KUKA KRL program: EPS_2_251455_MH64A_A_20251003045107.src

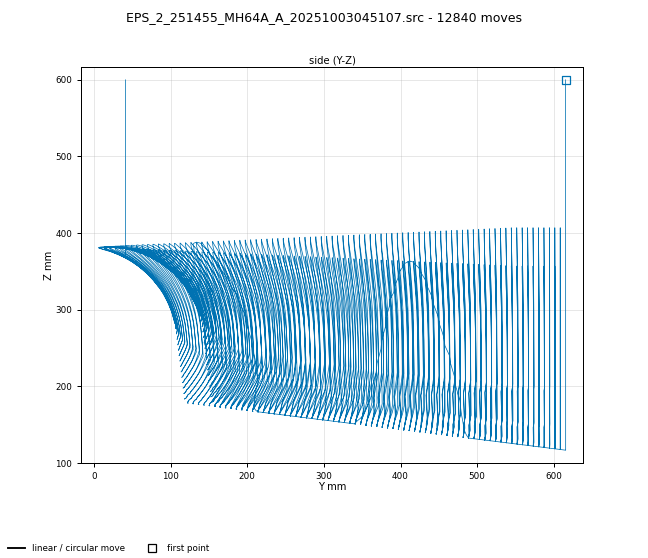
[picture p0: tool path of EPS_2_251455_MH64A_A_20251003045107.src, 12840 of 12842 moves have a stored position in this frame; points joined in program order, loops and branches not executed]
&ACCESS RVP
&REL 4
&COMMENT QRS 19112012
&PARAM EDITMASK = *
DEF PART()
EXT BAS (BAS_COMMAND :IN,REAL :IN )
INT I
BAS (#INITMOV,0 )

;KUKA QRS Post kuka4.cps  Date:22-06-2017 !

File_ID=2880

QRS_PRE_INIT()

;Init var - Until changes are made in qrs_pre_init
Outlet_Square_prg=0
Inlet_1_Square_prg=0
Inlet_2_Square_prg=0
Inlet_3_Square_prg=0
Inlet_4_Square_prg=0
Inlet_5_Square_prg=0

Outlet_1={X 0.000, Y 546.330, Z 306.500, B 0.000, E1 0.000 }
Inlet_1={X 0.000, Y 549.890, Z 256.500, B 0.000, E1 175.000 }
Outlet_1_type=201
Inlet_1_type=201
;QRS#1=Sidecore dimensions
;QRS#2=200-8" PVC SDR 35
;QRS#3=200-8" PVC SDR 35
;QRS#4=
;QRS#5=
;QRS#6=
;QRS#7=
;QRS#8=
;QRS#9=12-08 PSX
;QRS#10=12-08 PSX
;QRS#11=
;QRS#12=
;QRS#13=
;QRS#14=
;QRS#15=
;QRS#16=1220x127x686 2,25'
;QRS#17=EPS Height
;QRS#18=407
;QRS#19=*
;QRS#20= UPDATED VERSION 22-06-2017
;QRS#21=*
Outlet_Square=0100
Inlet_1_Square=0100
Inlet_2_Square=0
Inlet_3_Square=0
Inlet_4_Square=0
Inlet_5_Square=0
Mill_Square=1
Outlet_Square_Prg=204
Inlet_1_Square_prg=204

QRS_INIT()

$ADVANCE=5

; T1
PTP {E1 173.652,E2 173.652}
PTP {X 0,Y 615.443,A -85,B 0,C 180,E1 173.652,E2 173.652,E3 0,E4 0,E5 0,E6 0}
QRS_SPEED_INIT()
LIN {X 0,Y 615.443,Z 600,A -85,B 0,C 180,E1 173.652,E2 173.652,E3 0,E4 0,E5 0,E6 0} C_VEL
LIN {X 0,Y 615.443,Z 126.875,A -85,B 0,C 180,E1 173.652,E2 173.652} C_VEL
LIN {X 0,Y 615.443,Z 118.696,A -85,B 0,C 180,E1 173.652,E2 173.652} C_VEL
LIN {X 0,Y 615.432,Z 116.696,A -85,B 0,C 180,E1 173.465,E2 173.465} C_VEL
LIN {X 0,Y 615.432,Z 116.696,A -85,B 0,C 180,E1 171.462,E2 171.462} C_VEL
LIN {X 0,Y 615.436,Z 116.697,A -85,B 0,C 180,E1 169.136,E2 169.136} C_VEL
LIN {X 0,Y 615.468,Z 116.699,A -85,B 0,C 180,E1 166.798,E2 166.798} C_VEL
LIN {X 0,Y 615.467,Z 116.692,A -85,B 0,C 180,E1 164.094,E2 164.094} C_VEL
LIN {X 0,Y 615.458,Z 116.692,A -85,B 0,C 180,E1 162.042,E2 162.042} C_VEL
LIN {X 0,Y 615.45,Z 116.692,A -85,B 0,C 180,E1 159.966,E2 159.966} C_VEL
LIN {X 0,Y 615.442,Z 116.694,A -85,B 0,C 180,E1 157.664,E2 157.664} C_VEL
LIN {X 0,Y 615.491,Z 116.7,A -85,B 0,C 180,E1 155.008,E2 155.008} C_VEL
LIN {X 0,Y 615.495,Z 116.694,A -85,B 0,C 180,E1 152.823,E2 152.823} C_VEL
LIN {X 0,Y 615.456,Z 116.69,A -85,B 0,C 180,E1 150.21,E2 150.21} C_VEL
LIN {X 0,Y 615.457,Z 116.696,A -85,B 0,C 180,E1 147.674,E2 147.674} C_VEL
LIN {X 0,Y 615.496,Z 116.697,A -85,B 0,C 180,E1 145.185,E2 145.185} C_VEL
LIN {X 0,Y 615.489,Z 116.686,A -85,B 0,C 180,E1 142.758,E2 142.758} C_VEL
LIN {X 0,Y 615.454,Z 116.692,A -85,B 0,C 180,E1 140.247,E2 140.247} C_VEL
LIN {X 0,Y 615.489,Z 116.699,A -85,B 0,C 180,E1 137.647,E2 137.647} C_VEL
LIN {X 0,Y 615.492,Z 116.684,A -85,B 0,C 180,E1 134.932,E2 134.932} C_VEL
LIN {X 0,Y 615.47,Z 116.696,A -85,B 0,C 180,E1 132.078,E2 132.078} C_VEL
LIN {X 0,Y 615.493,Z 116.683,A -85,B 0,C 180,E1 129.062,E2 129.062} C_VEL
LIN {X 0,Y 615.467,Z 116.693,A -85,B 0,C 180,E1 126.426,E2 126.426} C_VEL
LIN {X 0,Y 615.485,Z 116.688,A -85,B 0,C 180,E1 123.533,E2 123.533} C_VEL
LIN {X 0,Y 615.473,Z 116.687,A -85,B 0,C 180,E1 120.921,E2 120.921} C_VEL
LIN {X 0,Y 615.481,Z 116.696,A -85,B 0,C 180,E1 118.448,E2 118.448} C_VEL
LIN {X 0,Y 615.487,Z 116.684,A -85,B 0,C 180,E1 115.568,E2 115.568} C_VEL
LIN {X 0,Y 615.474,Z 116.751,A -85,B 0,C 180,E1 112.979,E2 112.979} C_VEL
LIN {X 0,Y 615.47,Z 132.079,A -85,B 0,C 180,E1 110.294,E2 110.294} C_VEL
LIN {X 0,Y 615.477,Z 146.431,A -85,B 0,C 180,E1 107.807,E2 107.807} C_VEL
LIN {X 0,Y 615.434,Z 252.88,A -85,B 0,C 180,E1 106.545,E2 106.545} C_VEL
LIN {X 0,Y 615.441,Z 266.052,A -85,B 0,C 180,E1 106.255,E2 106.255} C_VEL
LIN {X 0,Y 615.481,Z 279.193,A -85,B 0,C 180,E1 105.821,E2 105.821} C_VEL
LIN {X 0,Y 615.47,Z 290.561,A -85,B 0,C 180,E1 105.312,E2 105.312} C_VEL
LIN {X 0,Y 615.475,Z 302.26,A -85,B 0,C 180,E1 104.634,E2 104.634} C_VEL
LIN {X 0,Y 615.498,Z 312.734,A -85,B 0,C 180,E1 103.874,E2 103.874} C_VEL
LIN {X 0,Y 615.497,Z 322.104,A -85,B 0,C 180,E1 103.034,E2 103.034} C_VEL
LIN {X 0,Y 615.497,Z 331.132,A -85,B 0,C 180,E1 102.028,E2 102.028} C_VEL
LIN {X 0,Y 615.497,Z 337.241,A -85,B 0,C 180,E1 101.193,E2 101.193} C_VEL
LIN {X 0,Y 615.497,Z 343.213,A -85,B 0,C 180,E1 100.195,E2 100.195} C_VEL
LIN {X 0,Y 615.496,Z 347.904,A -85,B 0,C 180,E1 99.199,E2 99.199} C_VEL
LIN {X 0,Y 615.496,Z 351.467,A -85,B 0,C 180,E1 98.206,E2 98.206} C_VEL
LIN {X 0,Y 615.496,Z 354.018,A -85,B 0,C 180,E1 97.216,E2 97.216} C_VEL
LIN {X 0,Y 615.495,Z 355.21,A -85,B 0,C 180,E1 96.557,E2 96.557} C_VEL
LIN {X 0,Y 615.499,Z 355.969,A -85,B 0,C 180,E1 95.899,E2 95.899} C_VEL
LIN {X 0,Y 615.498,Z 356.306,A -85,B 0,C 180,E1 94.585,E2 94.585} C_VEL
LIN {X 0,Y 615.497,Z 355.907,A -85,B 0,C 180,E1 93.929,E2 93.929} C_VEL
LIN {X 0,Y 615.496,Z 353.854,A -85,B 0,C 180,E1 92.618,E2 92.618} C_VEL
LIN {X 0,Y 615.498,Z 351.251,A -85,B 0,C 180,E1 91.636,E2 91.636} C_VEL
LIN {X 0,Y 615.496,Z 347.662,A -85,B 0,C 180,E1 90.655,E2 90.655} C_VEL
LIN {X 0,Y 615.495,Z 342.984,A -85,B 0,C 180,E1 89.673,E2 89.673} C_VEL
LIN {X 0,Y 615.497,Z 335.969,A -85,B 0,C 180,E1 88.528,E2 88.528} C_VEL
LIN {X 0,Y 615.496,Z 328.361,A -85,B 0,C 180,E1 87.547,E2 87.547} C_VEL
LIN {X 0,Y 615.498,Z 318.831,A -85,B 0,C 180,E1 86.564,E2 86.564} C_VEL
LIN {X 0,Y 615.498,Z 309.005,A -85,B 0,C 180,E1 85.744,E2 85.744} C_VEL
LIN {X 0,Y 615.461,Z 297.922,A -85,B 0,C 180,E1 85.006,E2 85.006} C_VEL
LIN {X 0,Y 615.479,Z 287.084,A -85,B 0,C 180,E1 84.431,E2 84.431} C_VEL
LIN {X 0,Y 615.476,Z 275.241,A -85,B 0,C 180,E1 83.942,E2 83.942} C_VEL
LIN {X 0,Y 615.447,Z 263.329,A -85,B 0,C 180,E1 83.582,E2 83.582} C_VEL
LIN {X 0,Y 615.441,Z 249.767,A -85,B 0,C 180,E1 83.32,E2 83.32} C_VEL
LIN {X 0,Y 615.485,Z 146.439,A -85,B 0,C 180,E1 82.104,E2 82.104} C_VEL
LIN {X 0,Y 615.49,Z 130.22,A -85,B 0,C 180,E1 79.294,E2 79.294} C_VEL
LIN {X 0,Y 615.467,Z 116.69,A -85,B 0,C 180,E1 76.883,E2 76.883} C_VEL
LIN {X 0,Y 615.489,Z 116.688,A -85,B 0,C 180,E1 74.096,E2 74.096} C_VEL
LIN {X 0,Y 615.468,Z 116.696,A -85,B 0,C 180,E1 71.354,E2 71.354} C_VEL
LIN {X 0,Y 615.49,Z 116.683,A -85,B 0,C 180,E1 68.569,E2 68.569} C_VEL
LIN {X 0,Y 615.484,Z 116.699,A -85,B 0,C 180,E1 65.729,E2 65.729} C_VEL
LIN {X 0,Y 615.466,Z 116.688,A -85,B 0,C 180,E1 62.96,E2 62.96} C_VEL
LIN {X 0,Y 615.494,Z 116.696,A -85,B 0,C 180,E1 60.205,E2 60.205} C_VEL
LIN {X 0,Y 615.457,Z 116.693,A -85,B 0,C 180,E1 57.542,E2 57.542} C_VEL
LIN {X 0,Y 615.463,Z 116.689,A -85,B 0,C 180,E1 55.185,E2 55.185} C_VEL
LIN {X 0,Y 615.496,Z 116.687,A -85,B 0,C 180,E1 52.76,E2 52.76} C_VEL
LIN {X 0,Y 615.457,Z 116.695,A -85,B 0,C 180,E1 49.915,E2 49.915} C_VEL
LIN {X 0,Y 615.449,Z 116.692,A -85,B 0,C 180,E1 47.645,E2 47.645} C_VEL
LIN {X 0,Y 615.497,Z 116.688,A -85,B 0,C 180,E1 44.934,E2 44.934} C_VEL
LIN {X 0,Y 615.449,Z 116.695,A -85,B 0,C 180,E1 42.078,E2 42.078} C_VEL
LIN {X 0,Y 615.444,Z 116.693,A -85,B 0,C 180,E1 39.754,E2 39.754} C_VEL
LIN {X 0,Y 615.49,Z 116.698,A -85,B 0,C 180,E1 36.939,E2 36.939} C_VEL
LIN {X 0,Y 615.439,Z 116.694,A -85,B 0,C 180,E1 34.025,E2 34.025} C_VEL
LIN {X 0,Y 615.487,Z 116.7,A -85,B 0,C 180,E1 31.088,E2 31.088} C_VEL
LIN {X 0,Y 615.439,Z 116.697,A -85,B 0,C 180,E1 28.445,E2 28.445} C_VEL
LIN {X 0,Y 615.435,Z 116.697,A -85,B 0,C 180,E1 26.447,E2 26.447} C_VEL
LIN {X 0,Y 615.442,Z 116.694,A -85,B 0,C 180,E1 24.002,E2 24.002} C_VEL
LIN {X 0,Y 615.498,Z 116.696,A -85,B 0,C 180,E1 21.432,E2 21.432} C_VEL
LIN {X 0,Y 615.427,Z 116.697,A -85,B 0,C 180,E1 18.592,E2 18.592} C_VEL
LIN {X 0,Y 615.464,Z 116.695,A -85,B 0,C 180,E1 15.906,E2 15.906} C_VEL
LIN {X 0,Y 615.449,Z 116.699,A -85,B 0,C 180,E1 13.202,E2 13.202} C_VEL
LIN {X 0,Y 615.422,Z 116.699,A -85,B 0,C 180,E1 10.864,E2 10.864} C_VEL
LIN {X 0,Y 615.423,Z 116.699,A -85,B 0,C 180,E1 8.538,E2 8.538} C_VEL
LIN {X 0,Y 615.496,Z 116.698,A -85,B 0,C 180,E1 5.899,E2 5.899} C_VEL
LIN {X 0,Y 615.424,Z 116.7,A -85,B 0,C 180,E1 3.273,E2 3.273} C_VEL
LIN {X 0,Y 615.422,Z 116.7,A -85,B 0,C 180,E1 1.309,E2 1.309} C_VEL
LIN {X 0,Y 615.423,Z 116.7,A -85,B 0,C 180,E1 -0.654,E2 -0.654} C_VEL
LIN {X 0,Y 615.424,Z 116.699,A -85,B 0,C 180,E1 -2.618,E2 -2.618} C_VEL
LIN {X 0,Y 615.425,Z 116.699,A -85,B 0,C 180,E1 -4.585,E2 -4.585} C_VEL
LIN {X 0,Y 615.425,Z 116.698,A -85,B 0,C 180,E1 -6.557,E2 -6.557} C_VEL
LIN {X 0,Y 615.425,Z 116.698,A -85,B 0,C 180,E1 -8.537,E2 -8.537} C_VEL
LIN {X 0,Y 615.426,Z 116.698,A -85,B 0,C 180,E1 -10.866,E2 -10.866} C_VEL
LIN {X 0,Y 615.454,Z 116.699,A -85,B 0,C 180,E1 -13.202,E2 -13.202} C_VEL
LIN {X 0,Y 615.465,Z 116.694,A -85,B 0,C 180,E1 -15.906,E2 -15.906} C_VEL
LIN {X 0,Y 615.454,Z 116.694,A -85,B 0,C 180,E1 -17.958,E2 -17.958} C_VEL
LIN {X 0,Y 615.433,Z 116.697,A -85,B 0,C 180,E1 -20.547,E2 -20.547} C_VEL
LIN {X 0,Y 615.454,Z 116.698,A -85,B 0,C 180,E1 -22.846,E2 -22.846} C_VEL
LIN {X 0,Y 615.464,Z 116.692,A -85,B 0,C 180,E1 -25.717,E2 -25.717} C_VEL
LIN {X 0,Y 615.446,Z 116.693,A -85,B 0,C 180,E1 -27.917,E2 -27.917} C_VEL
LIN {X 0,Y 615.439,Z 116.695,A -85,B 0,C 180,E1 -30.163,E2 -30.163} C_VEL
LIN {X 0,Y 615.451,Z 116.697,A -85,B 0,C 180,E1 -32.46,E2 -32.46} C_VEL
LIN {X 0,Y 615.494,Z 116.7,A -85,B 0,C 180,E1 -34.815,E2 -34.815} C_VEL
LIN {X 0,Y 615.488,Z 116.688,A -85,B 0,C 180,E1 -37.242,E2 -37.242} C_VEL
LIN {X 0,Y 615.446,Z 116.693,A -85,B 0,C 180,E1 -39.754,E2 -39.754} C_VEL
LIN {X 0,Y 615.472,Z 116.698,A -85,B 0,C 180,E1 -42.354,E2 -42.354} C_VEL
LIN {X 0,Y 615.492,Z 116.686,A -85,B 0,C 180,E1 -45.068,E2 -45.068} C_VEL
LIN {X 0,Y 615.452,Z 116.692,A -85,B 0,C 180,E1 -47.646,E2 -47.646} C_VEL
LIN {X 0,Y 615.49,Z 116.699,A -85,B 0,C 180,E1 -50.251,E2 -50.251} C_VEL
LIN {X 0,Y 615.475,Z 116.687,A -85,B 0,C 180,E1 -53.065,E2 -53.065} C_VEL
LIN {X 0,Y 615.459,Z 116.69,A -85,B 0,C 180,E1 -55.304,E2 -55.304} C_VEL
LIN {X 0,Y 615.464,Z 116.695,A -85,B 0,C 180,E1 -57.673,E2 -57.673} C_VEL
LIN {X 0,Y 615.489,Z 116.686,A -85,B 0,C 180,E1 -60.595,E2 -60.595} C_VEL
LIN {X 0,Y 615.468,Z 116.688,A -85,B 0,C 180,E1 -62.959,E2 -62.959} C_VEL
LIN {X 0,Y 615.483,Z 116.7,A -85,B 0,C 180,E1 -65.729,E2 -65.729} C_VEL
LIN {X 0,Y 615.464,Z 116.83,A -85,B 0,C 180,E1 -67.067,E2 -67.067} C_VEL
LIN {X 0,Y 615.465,Z 136.774,A -85,B 0,C 180,E1 -69.707,E2 -69.707} C_VEL
LIN {X 0,Y 615.485,Z 158.677,A -85,B 0,C 180,E1 -72.559,E2 -72.559} C_VEL
LIN {X 0,Y 615.469,Z 179.898,A -85,B 0,C 180,E1 -75.282,E2 -75.282} C_VEL
LIN {X 0,Y 615.452,Z 194.307,A -85,B 0,C 180,E1 -77.114,E2 -77.114} C_VEL
LIN {X 0,Y 615.488,Z 302.873,A -85,B 0,C 180,E1 -78.411,E2 -78.411} C_VEL
LIN {X 0,Y 615.477,Z 315.374,A -85,B 0,C 180,E1 -78.682,E2 -78.682} C_VEL
LIN {X 0,Y 615.488,Z 328.617,A -85,B 0,C 180,E1 -79.113,E2 -79.113} C_VEL
LIN {X 0,Y 615.477,Z 340.493,A -85,B 0,C 180,E1 -79.64,E2 -79.64} C_VEL
LIN {X 0,Y 615.494,Z 352.005,A -85,B 0,C 180,E1 -80.305,E2 -80.305} C_VEL
LIN {X 0,Y 615.499,Z 362.35,A -85,B 0,C 180,E1 -81.051,E2 -81.051} C_VEL
LIN {X 0,Y 615.497,Z 370.819,A -85,B 0,C 180,E1 -81.795,E2 -81.795} C_VEL
LIN {X 0,Y 615.498,Z 378.612,A -85,B 0,C 180,E1 -82.62,E2 -82.62} C_VEL
LIN {X 0,Y 615.496,Z 386.208,A -85,B 0,C 180,E1 -83.609,E2 -83.609} C_VEL
LIN {X 0,Y 615.498,Z 393.208,A -85,B 0,C 180,E1 -84.76,E2 -84.76} C_VEL
LIN {X 0,Y 615.494,Z 397.854,A -85,B 0,C 180,E1 -85.744,E2 -85.744} C_VEL
LIN {X 0,Y 615.494,Z 401.401,A -85,B 0,C 180,E1 -86.728,E2 -86.728} C_VEL
LIN {X 0,Y 615.497,Z 403.234,A -85,B 0,C 180,E1 -87.383,E2 -87.383} C_VEL
LIN {X 0,Y 615.5,Z 404.608,A -85,B 0,C 180,E1 -88.038,E2 -88.038} C_VEL
LIN {X 0,Y 615.496,Z 406.174,A -85,B 0,C 180,E1 -89.346,E2 -89.346} C_VEL
LIN {X 0,Y 615.494,Z 406.389,A -85,B 0,C 180,E1 -90.001,E2 -90.001} C_VEL
LIN {X 0,Y 615.495,Z 405.579,A -85,B 0,C 180,E1 -91.309,E2 -91.309} C_VEL
LIN {X 0,Y 615.5,Z 404.606,A -85,B 0,C 180,E1 -91.964,E2 -91.964} C_VEL
LIN {X 0,Y 615.497,Z 403.231,A -85,B 0,C 180,E1 -92.618,E2 -92.618} C_VEL
LIN {X 0,Y 615.496,Z 400.348,A -85,B 0,C 180,E1 -93.601,E2 -93.601} C_VEL
LIN {X 0,Y 615.498,Z 396.439,A -85,B 0,C 180,E1 -94.585,E2 -94.585} C_VEL
LIN {X 0,Y 615.499,Z 391.402,A -85,B 0,C 180,E1 -95.57,E2 -95.57} C_VEL
LIN {X 0,Y 615.497,Z 384.869,A -85,B 0,C 180,E1 -96.583,E2 -96.583} C_VEL
LIN {X 0,Y 615.497,Z 377.129,A -85,B 0,C 180,E1 -97.546,E2 -97.546} C_VEL
LIN {X 0,Y 615.498,Z 369.04,A -85,B 0,C 180,E1 -98.372,E2 -98.372} C_VEL
LIN {X 0,Y 615.499,Z 359.161,A -85,B 0,C 180,E1 -99.199,E2 -99.199} C_VEL
LIN {X 0,Y 615.488,Z 347.974,A -85,B 0,C 180,E1 -99.946,E2 -99.946} C_VEL
LIN {X 0,Y 615.482,Z 337.014,A -85,B 0,C 180,E1 -100.527,E2 -100.527} C_VEL
LIN {X 0,Y 615.48,Z 324.483,A -85,B 0,C 180,E1 -101.04,E2 -101.04} C_VEL
LIN {X 0,Y 615.479,Z 312.047,A -85,B 0,C 180,E1 -101.402,E2 -101.402} C_VEL
LIN {X 0,Y 615.493,Z 298.432,A -85,B 0,C 180,E1 -101.652,E2 -101.652} C_VEL
LIN {X 0,Y 615.452,Z 194.297,A -85,B 0,C 180,E1 -102.888,E2 -102.888} C_VEL
LIN {X 0,Y 615.494,Z 171.93,A -85,B 0,C 180,E1 -105.735,E2 -105.735} C_VEL
LIN {X 0,Y 615.456,Z 151.012,A -85,B 0,C 180,E1 -108.435,E2 -108.435} C_VEL
LIN {X 0,Y 615.488,Z 130.779,A -85,B 0,C 180,E1 -111.081,E2 -111.081} C_VEL
LIN {X 0,Y 615.465,Z 116.689,A -85,B 0,C 180,E1 -112.979,E2 -112.979} C_VEL
LIN {X 0,Y 615.49,Z 116.69,A -85,B 0,C 180,E1 -115.716,E2 -115.716} C_VEL
LIN {X 0,Y 615.465,Z 116.695,A -85,B 0,C 180,E1 -118.446,E2 -118.446} C_VEL
LIN {X 0,Y 615.477,Z 116.686,A -85,B 0,C 180,E1 -121.084,E2 -121.084} C_VEL
LIN {X 0,Y 615.477,Z 116.698,A -85,B 0,C 180,E1 -124.023,E2 -124.023} C_VEL
LIN {X 0,Y 615.454,Z 116.693,A -85,B 0,C 180,E1 -126.427,E2 -126.427} C_VEL
LIN {X 0,Y 615.492,Z 116.686,A -85,B 0,C 180,E1 -129.062,E2 -129.062} C_VEL
LIN {X 0,Y 615.494,Z 116.698,A -85,B 0,C 180,E1 -131.473,E2 -131.473} C_VEL
LIN {X 0,Y 615.449,Z 116.694,A -85,B 0,C 180,E1 -134.153,E2 -134.153} C_VEL
LIN {X 0,Y 615.488,Z 116.69,A -85,B 0,C 180,E1 -136.953,E2 -136.953} C_VEL
LIN {X 0,Y 615.479,Z 116.701,A -85,B 0,C 180,E1 -139.393,E2 -139.393} C_VEL
LIN {X 0,Y 615.44,Z 116.695,A -85,B 0,C 180,E1 -141.994,E2 -141.994} C_VEL
LIN {X 0,Y 615.451,Z 116.693,A -85,B 0,C 180,E1 -144.382,E2 -144.382} C_VEL
LIN {X 0,Y 615.489,Z 116.693,A -85,B 0,C 180,E1 -146.764,E2 -146.764} C_VEL
LIN {X 0,Y 615.477,Z 116.701,A -85,B 0,C 180,E1 -149.08,E2 -149.08} C_VEL
LIN {X 0,Y 615.434,Z 116.697,A -85,B 0,C 180,E1 -151.559,E2 -151.559} C_VEL
LIN {X 0,Y 615.433,Z 116.697,A -85,B 0,C 180,E1 -153.553,E2 -153.553} C_VEL
LIN {X 0,Y 615.441,Z 116.695,A -85,B 0,C 180,E1 -156.001,E2 -156.001} C_VEL
LIN {X 0,Y 615.498,Z 116.698,A -85,B 0,C 180,E1 -158.568,E2 -158.568} C_VEL
LIN {X 0,Y 615.423,Z 116.698,A -85,B 0,C 180,E1 -161.413,E2 -161.413} C_VEL
LIN {X 0,Y 615.463,Z 116.697,A -85,B 0,C 180,E1 -164.094,E2 -164.094} C_VEL
LIN {X 0,Y 615.442,Z 116.7,A -85,B 0,C 180,E1 -166.798,E2 -166.798} C_VEL
LIN {X 0,Y 615.416,Z 116.7,A -85,B 0,C 180,E1 -169.145,E2 -169.145} C_VEL
LIN {X 0,Y 615.419,Z 116.7,A -85,B 0,C 180,E1 -171.462,E2 -171.462} C_VEL
LIN {X 0,Y 615.498,Z 116.7,A -85,B 0,C 180,E1 -174.102,E2 -174.102} C_VEL
LIN {X 0,Y 615.426,Z 116.699,A -85,B 0,C 180,E1 -176.727,E2 -176.727} C_VEL
LIN {X 0,Y 615.426,Z 116.698,A -85,B 0,C 180,E1 -178.691,E2 -178.691} C_VEL
LIN {X 0,Y 615.428,Z 116.698,A -85,B 0,C 180,E1 -180.654,E2 -180.654} C_VEL
LIN {X 0,Y 615.429,Z 116.697,A -85,B 0,C 180,E1 -182.618,E2 -182.618} C_VEL
LIN {X 0,Y 615.43,Z 116.697,A -85,B 0,C 180,E1 -184.585,E2 -184.585} C_VEL
LIN {X 0,Y 615.432,Z 116.696,A -85,B 0,C 180,E1 -186.535,E2 -186.535} C_VEL
LIN {X 0,Y 614.764,Z 116.846,A -85,B 0,C 180,E1 -187.081,E2 -187.081} C_VEL
LIN {X 0,Y 611.939,Z 117.258,A -85,B 0,C 180,E1 -187.967,E2 -187.967} C_VEL
LIN {X 0,Y 609.554,Z 117.569,A -85,B 0,C 180,E1 -188.68,E2 -188.68} C_VEL
LIN {X 0,Y 608.526,Z 117.686,A -85,B 0,C 180,E1 -189.23,E2 -189.23} C_VEL
LIN {X 0,Y 608.439,Z 117.694,A -85,B 0,C 180,E1 -189.416,E2 -189.416} C_VEL
LIN {X 0,Y 608.446,Z 117.691,A -85,B 0,C 180,E1 -192,E2 -192} C_VEL
LIN {X 0,Y 608.407,Z 117.694,A -85,B 0,C 180,E1 -194.722,E2 -194.722} C_VEL
LIN {X 0,Y 608.45,Z 117.695,A -85,B 0,C 180,E1 -197.477,E2 -197.477} C_VEL
LIN {X 0,Y 608.426,Z 117.691,A -85,B 0,C 180,E1 -200.276,E2 -200.276} C_VEL
LIN {X 0,Y 608.428,Z 117.692,A -85,B 0,C 180,E1 -202.47,E2 -202.47} C_VEL
LIN {X 0,Y 608.451,Z 117.694,A -85,B 0,C 180,E1 -205.301,E2 -205.301} C_VEL
LIN {X 0,Y 608.44,Z 117.691,A -85,B 0,C 180,E1 -207.519,E2 -207.519} C_VEL
LIN {X 0,Y 608.421,Z 117.692,A -85,B 0,C 180,E1 -209.964,E2 -209.964} C_VEL
LIN {X 0,Y 608.445,Z 117.694,A -85,B 0,C 180,E1 -212.52,E2 -212.52} C_VEL
LIN {X 0,Y 608.434,Z 117.692,A -85,B 0,C 180,E1 -215.279,E2 -215.279} C_VEL
LIN {X 0,Y 608.452,Z 117.688,A -85,B 0,C 180,E1 -217.748,E2 -217.748} C_VEL
LIN {X 0,Y 608.442,Z 117.696,A -85,B 0,C 180,E1 -220.328,E2 -220.328} C_VEL
LIN {X 0,Y 608.468,Z 117.686,A -85,B 0,C 180,E1 -223.309,E2 -223.309} C_VEL
LIN {X 0,Y 608.459,Z 117.694,A -85,B 0,C 180,E1 -226.13,E2 -226.13} C_VEL
LIN {X 0,Y 608.458,Z 117.689,A -85,B 0,C 180,E1 -228.824,E2 -228.824} C_VEL
LIN {X 0,Y 608.435,Z 117.691,A -85,B 0,C 180,E1 -231.409,E2 -231.409} C_VEL
LIN {X 0,Y 608.45,Z 117.697,A -85,B 0,C 180,E1 -233.955,E2 -233.955} C_VEL
LIN {X 0,Y 608.454,Z 117.692,A -85,B 0,C 180,E1 -236.328,E2 -236.328} C_VEL
LIN {X 0,Y 608.449,Z 117.688,A -85,B 0,C 180,E1 -238.733,E2 -238.733} C_VEL
LIN {X 0,Y 608.466,Z 117.69,A -85,B 0,C 180,E1 -241.382,E2 -241.382} C_VEL
LIN {X 0,Y 608.445,Z 117.695,A -85,B 0,C 180,E1 -243.964,E2 -243.964} C_VEL
LIN {X 0,Y 608.464,Z 117.689,A -85,B 0,C 180,E1 -246.155,E2 -246.155} C_VEL
LIN {X 0,Y 608.452,Z 117.731,A -85,B 0,C 180,E1 -246.966,E2 -246.966} C_VEL
LIN {X 0,Y 608.45,Z 132.208,A -85,B 0,C 180,E1 -249.524,E2 -249.524} C_VEL
LIN {X 0,Y 608.457,Z 146.656,A -85,B 0,C 180,E1 -252.046,E2 -252.046} C_VEL
LIN {X 0,Y 608.489,Z 253.763,A -85,B 0,C 180,E1 -253.336,E2 -253.336} C_VEL
LIN {X 0,Y 608.477,Z 267.45,A -85,B 0,C 180,E1 -253.65,E2 -253.65} C_VEL
LIN {X 0,Y 608.51,Z 279.993,A -85,B 0,C 180,E1 -254.079,E2 -254.079} C_VEL
LIN {X 0,Y 608.472,Z 291.201,A -85,B 0,C 180,E1 -254.594,E2 -254.594} C_VEL
LIN {X 0,Y 608.469,Z 302.853,A -85,B 0,C 180,E1 -255.279,E2 -255.279} C_VEL
LIN {X 0,Y 608.482,Z 312.457,A -85,B 0,C 180,E1 -255.98,E2 -255.98} C_VEL
LIN {X 0,Y 608.476,Z 321.835,A -85,B 0,C 180,E1 -256.813,E2 -256.813} C_VEL
LIN {X 0,Y 608.462,Z 331.024,A -85,B 0,C 180,E1 -257.831,E2 -257.831} C_VEL
LIN {X 0,Y 608.46,Z 339.01,A -85,B 0,C 180,E1 -258.937,E2 -258.937} C_VEL
LIN {X 0,Y 608.438,Z 345.106,A -85,B 0,C 180,E1 -260.022,E2 -260.022} C_VEL
LIN {X 0,Y 608.446,Z 349.518,A -85,B 0,C 180,E1 -261.029,E2 -261.029} C_VEL
LIN {X 0,Y 608.424,Z 352.836,A -85,B 0,C 180,E1 -262.032,E2 -262.032} C_VEL
LIN {X 0,Y 608.422,Z 354.479,A -85,B 0,C 180,E1 -262.7,E2 -262.7} C_VEL
LIN {X 0,Y 608.448,Z 355.762,A -85,B 0,C 180,E1 -263.397,E2 -263.397} C_VEL
LIN {X 0,Y 608.435,Z 356.535,A -85,B 0,C 180,E1 -264.032,E2 -264.032} C_VEL
LIN {X 0,Y 608.431,Z 356.932,A -85,B 0,C 180,E1 -265.362,E2 -265.362} C_VEL
LIN {X 0,Y 608.434,Z 356.56,A -85,B 0,C 180,E1 -266.025,E2 -266.025} C_VEL
LIN {X 0,Y 608.422,Z 355.77,A -85,B 0,C 180,E1 -266.688,E2 -266.688} C_VEL
LIN {X 0,Y 608.445,Z 352.955,A -85,B 0,C 180,E1 -268.014,E2 -268.014} C_VEL
LIN {X 0,Y 608.426,Z 349.723,A -85,B 0,C 180,E1 -269.007,E2 -269.007} C_VEL
LIN {X 0,Y 608.436,Z 345.44,A -85,B 0,C 180,E1 -269.999,E2 -269.999} C_VEL
LIN {X 0,Y 608.452,Z 338.98,A -85,B 0,C 180,E1 -271.158,E2 -271.158} C_VEL
LIN {X 0,Y 608.454,Z 331.911,A -85,B 0,C 180,E1 -272.151,E2 -272.151} C_VEL
LIN {X 0,Y 608.459,Z 323.126,A -85,B 0,C 180,E1 -273.144,E2 -273.144} C_VEL
LIN {X 0,Y 608.469,Z 314.15,A -85,B 0,C 180,E1 -273.973,E2 -273.973} C_VEL
LIN {X 0,Y 608.481,Z 304.239,A -85,B 0,C 180,E1 -274.72,E2 -274.72} C_VEL
LIN {X 0,Y 608.466,Z 293.29,A -85,B 0,C 180,E1 -275.384,E2 -275.384} C_VEL
LIN {X 0,Y 608.528,Z 281.059,A -85,B 0,C 180,E1 -275.966,E2 -275.966} C_VEL
LIN {X 0,Y 608.497,Z 268.623,A -85,B 0,C 180,E1 -276.407,E2 -276.407} C_VEL
LIN {X 0,Y 608.497,Z 255.904,A -85,B 0,C 180,E1 -276.715,E2 -276.715} C_VEL
LIN {X 0,Y 608.511,Z 237.722,A -85,B 0,C 180,E1 -276.964,E2 -276.964} C_VEL
LIN {X 0,Y 608.462,Z 146.624,A -85,B 0,C 180,E1 -278.05,E2 -278.05} C_VEL
LIN {X 0,Y 608.467,Z 131.734,A -85,B 0,C 180,E1 -280.649,E2 -280.649} C_VEL
LIN {X 0,Y 608.439,Z 117.691,A -85,B 0,C 180,E1 -283.144,E2 -283.144} C_VEL
LIN {X 0,Y 608.461,Z 117.687,A -85,B 0,C 180,E1 -285.405,E2 -285.405} C_VEL
LIN {X 0,Y 608.446,Z 117.696,A -85,B 0,C 180,E1 -288.171,E2 -288.171} C_VEL
LIN {X 0,Y 608.448,Z 117.689,A -85,B 0,C 180,E1 -290.981,E2 -290.981} C_VEL
LIN {X 0,Y 608.472,Z 117.691,A -85,B 0,C 180,E1 -293.844,E2 -293.844} C_VEL
LIN {X 0,Y 608.439,Z 117.699,A -85,B 0,C 180,E1 -296.035,E2 -296.035} C_VEL
LIN {X 0,Y 608.451,Z 117.689,A -85,B 0,C 180,E1 -298.615,E2 -298.615} C_VEL
LIN {X 0,Y 608.458,Z 117.689,A -85,B 0,C 180,E1 -301.316,E2 -301.316} C_VEL
LIN {X 0,Y 608.473,Z 117.694,A -85,B 0,C 180,E1 -303.734,E2 -303.734} C_VEL
LIN {X 0,Y 608.438,Z 117.694,A -85,B 0,C 180,E1 -306.091,E2 -306.091} C_VEL
LIN {X 0,Y 608.426,Z 117.691,A -85,B 0,C 180,E1 -308.59,E2 -308.59} C_VEL
LIN {X 0,Y 608.467,Z 117.692,A -85,B 0,C 180,E1 -311.342,E2 -311.342} C_VEL
LIN {X 0,Y 608.446,Z 117.693,A -85,B 0,C 180,E1 -313.87,E2 -313.87} C_VEL
LIN {X 0,Y 608.463,Z 117.687,A -85,B 0,C 180,E1 -316.69,E2 -316.69} C_VEL
LIN {X 0,Y 608.445,Z 117.693,A -85,B 0,C 180,E1 -319.696,E2 -319.696} C_VEL
LIN {X 0,Y 608.48,Z 117.689,A -85,B 0,C 180,E1 -322.838,E2 -322.838} C_VEL
LIN {X 0,Y 608.45,Z 117.692,A -85,B 0,C 180,E1 -325.529,E2 -325.529} C_VEL
LIN {X 0,Y 608.428,Z 117.691,A -85,B 0,C 180,E1 -327.903,E2 -327.903} C_VEL
LIN {X 0,Y 608.436,Z 117.691,A -85,B 0,C 180,E1 -330.218,E2 -330.218} C_VEL
LIN {X 0,Y 608.481,Z 117.693,A -85,B 0,C 180,E1 -332.789,E2 -332.789} C_VEL
LIN {X 0,Y 608.42,Z 117.693,A -85,B 0,C 180,E1 -335.427,E2 -335.427} C_VEL
LIN {X 0,Y 608.456,Z 117.691,A -85,B 0,C 180,E1 -338.308,E2 -338.308} C_VEL
LIN {X 0,Y 608.409,Z 117.694,A -85,B 0,C 180,E1 -341.297,E2 -341.297} C_VEL
LIN {X 0,Y 608.426,Z 117.693,A -85,B 0,C 180,E1 -343.905,E2 -343.905} C_VEL
LIN {X 0,Y 608.434,Z 117.697,A -85,B 0,C 180,E1 -346.643,E2 -346.643} C_VEL
LIN {X 0,Y 608.404,Z 117.694,A -85,B 0,C 180,E1 -349.349,E2 -349.349} C_VEL
LIN {X 0,Y 608.462,Z 117.693,A -85,B 0,C 180,E1 -352.033,E2 -352.033} C_VEL
LIN {X 0,Y 608.416,Z 117.695,A -85,B 0,C 180,E1 -354.698,E2 -354.698} C_VEL
LIN {X 0,Y 608.417,Z 117.693,A -85,B 0,C 180,E1 -357.352,E2 -357.352} C_VEL
LIN {X 0,Y 608.465,Z 117.697,A -85,B 0,C 180,E1 -360,E2 -360} C_VEL
LIN {X 0,Y 608.419,Z 117.693,A -85,B 0,C 180,E1 -362.648,E2 -362.648} C_VEL
LIN {X 0,Y 608.42,Z 117.695,A -85,B 0,C 180,E1 -365.302,E2 -365.302} C_VEL
LIN {X 0,Y 608.464,Z 117.692,A -85,B 0,C 180,E1 -367.967,E2 -367.967} C_VEL
LIN {X 0,Y 608.422,Z 117.693,A -85,B 0,C 180,E1 -370.94,E2 -370.94} C_VEL
LIN {X 0,Y 608.437,Z 117.697,A -85,B 0,C 180,E1 -373.357,E2 -373.357} C_VEL
LIN {X 0,Y 608.427,Z 117.692,A -85,B 0,C 180,E1 -376.095,E2 -376.095} C_VEL
LIN {X 0,Y 608.429,Z 117.693,A -85,B 0,C 180,E1 -378.87,E2 -378.87} C_VEL
LIN {X 0,Y 608.457,Z 117.691,A -85,B 0,C 180,E1 -381.692,E2 -381.692} C_VEL
LIN {X 0,Y 608.423,Z 117.693,A -85,B 0,C 180,E1 -384.572,E2 -384.572} C_VEL
LIN {X 0,Y 608.484,Z 117.692,A -85,B 0,C 180,E1 -387.211,E2 -387.211} C_VEL
LIN {X 0,Y 608.414,Z 117.693,A -85,B 0,C 180,E1 -389.965,E2 -389.965} C_VEL
LIN {X 0,Y 608.431,Z 117.694,A -85,B 0,C 180,E1 -392.52,E2 -392.52} C_VEL
LIN {X 0,Y 608.429,Z 117.694,A -85,B 0,C 180,E1 -395.279,E2 -395.279} C_VEL
LIN {X 0,Y 608.443,Z 117.689,A -85,B 0,C 180,E1 -397.748,E2 -397.748} C_VEL
LIN {X 0,Y 608.429,Z 117.695,A -85,B 0,C 180,E1 -400.328,E2 -400.328} C_VEL
LIN {X 0,Y 608.463,Z 117.687,A -85,B 0,C 180,E1 -403.31,E2 -403.31} C_VEL
LIN {X 0,Y 608.449,Z 117.693,A -85,B 0,C 180,E1 -406.13,E2 -406.13} C_VEL
LIN {X 0,Y 608.458,Z 117.69,A -85,B 0,C 180,E1 -408.825,E2 -408.825} C_VEL
LIN {X 0,Y 608.428,Z 117.691,A -85,B 0,C 180,E1 -411.41,E2 -411.41} C_VEL
LIN {X 0,Y 608.442,Z 117.695,A -85,B 0,C 180,E1 -413.955,E2 -413.955} C_VEL
LIN {X 0,Y 608.465,Z 117.693,A -85,B 0,C 180,E1 -416.331,E2 -416.331} C_VEL
LIN {X 0,Y 608.474,Z 117.686,A -85,B 0,C 180,E1 -418.729,E2 -418.729} C_VEL
LIN {X 0,Y 608.453,Z 117.689,A -85,B 0,C 180,E1 -421.384,E2 -421.384} C_VEL
LIN {X 0,Y 608.441,Z 117.698,A -85,B 0,C 180,E1 -423.965,E2 -423.965} C_VEL
LIN {X 0,Y 608.471,Z 117.692,A -85,B 0,C 180,E1 -426.156,E2 -426.156} C_VEL
LIN {X 0,Y 608.467,Z 117.828,A -85,B 0,C 180,E1 -426.923,E2 -426.923} C_VEL
LIN {X 0,Y 608.584,Z 133.45,A -85,B 0,C 180,E1 -429.024,E2 -429.024} C_VEL
LIN {X 0,Y 608.522,Z 154.723,A -85,B 0,C 180,E1 -431.831,E2 -431.831} C_VEL
LIN {X 0,Y 608.49,Z 175.997,A -85,B 0,C 180,E1 -434.595,E2 -434.595} C_VEL
LIN {X 0,Y 608.449,Z 194.528,A -85,B 0,C 180,E1 -436.973,E2 -436.973} C_VEL
LIN {X 0,Y 608.546,Z 302.989,A -85,B 0,C 180,E1 -438.277,E2 -438.277} C_VEL
LIN {X 0,Y 608.512,Z 316.245,A -85,B 0,C 180,E1 -438.572,E2 -438.572} C_VEL
LIN {X 0,Y 608.514,Z 328.633,A -85,B 0,C 180,E1 -438.982,E2 -438.982} C_VEL
LIN {X 0,Y 608.499,Z 340.649,A -85,B 0,C 180,E1 -439.52,E2 -439.52} C_VEL
LIN {X 0,Y 608.484,Z 352.209,A -85,B 0,C 180,E1 -440.192,E2 -440.192} C_VEL
LIN {X 0,Y 608.485,Z 362.603,A -85,B 0,C 180,E1 -440.947,E2 -440.947} C_VEL
LIN {X 0,Y 608.475,Z 371.12,A -85,B 0,C 180,E1 -441.7,E2 -441.7} C_VEL
LIN {X 0,Y 608.47,Z 378.966,A -85,B 0,C 180,E1 -442.535,E2 -442.535} C_VEL
LIN {X 0,Y 608.46,Z 386.289,A -85,B 0,C 180,E1 -443.485,E2 -443.485} C_VEL
LIN {X 0,Y 608.451,Z 391.87,A -85,B 0,C 180,E1 -444.366,E2 -444.366} C_VEL
LIN {X 0,Y 608.432,Z 396.953,A -85,B 0,C 180,E1 -445.363,E2 -445.363} C_VEL
LIN {X 0,Y 608.449,Z 400.898,A -85,B 0,C 180,E1 -446.358,E2 -446.358} C_VEL
LIN {X 0,Y 608.425,Z 403.811,A -85,B 0,C 180,E1 -447.352,E2 -447.352} C_VEL
LIN {X 0,Y 608.445,Z 405.202,A -85,B 0,C 180,E1 -448.015,E2 -448.015} C_VEL
LIN {X 0,Y 608.438,Z 406.784,A -85,B 0,C 180,E1 -449.339,E2 -449.339} C_VEL
LIN {X 0,Y 608.434,Z 407,A -85,B 0,C 180,E1 -450.001,E2 -450.001} C_VEL
LIN {X 0,Y 608.448,Z 406.183,A -85,B 0,C 180,E1 -451.324,E2 -451.324} C_VEL
LIN {X 0,Y 608.445,Z 405.2,A -85,B 0,C 180,E1 -451.986,E2 -451.986} C_VEL
LIN {X 0,Y 608.425,Z 403.808,A -85,B 0,C 180,E1 -452.649,E2 -452.649} C_VEL
LIN {X 0,Y 608.449,Z 400.894,A -85,B 0,C 180,E1 -453.643,E2 -453.643} C_VEL
LIN {X 0,Y 608.432,Z 396.948,A -85,B 0,C 180,E1 -454.638,E2 -454.638} C_VEL
LIN {X 0,Y 608.438,Z 390.873,A -85,B 0,C 180,E1 -455.801,E2 -455.801} C_VEL
LIN {X 0,Y 608.462,Z 384.231,A -85,B 0,C 180,E1 -456.8,E2 -456.8} C_VEL
LIN {X 0,Y 608.456,Z 375.985,A -85,B 0,C 180,E1 -457.801,E2 -457.801} C_VEL
LIN {X 0,Y 608.472,Z 367.531,A -85,B 0,C 180,E1 -458.636,E2 -458.636} C_VEL
LIN {X 0,Y 608.479,Z 357.084,A -85,B 0,C 180,E1 -459.474,E2 -459.474} C_VEL
LIN {X 0,Y 608.489,Z 346.748,A -85,B 0,C 180,E1 -460.145,E2 -460.145} C_VEL
LIN {X 0,Y 608.519,Z 335.259,A -85,B 0,C 180,E1 -460.74,E2 -460.74} C_VEL
LIN {X 0,Y 608.528,Z 322.879,A -85,B 0,C 180,E1 -461.225,E2 -461.225} C_VEL
LIN {X 0,Y 608.544,Z 309.419,A -85,B 0,C 180,E1 -461.597,E2 -461.597} C_VEL
LIN {X 0,Y 608.553,Z 297.049,A -85,B 0,C 180,E1 -461.808,E2 -461.808} C_VEL
LIN {X 0,Y 608.438,Z 194.435,A -85,B 0,C 180,E1 -463.039,E2 -463.039} C_VEL
LIN {X 0,Y 608.51,Z 171.998,A -85,B 0,C 180,E1 -465.921,E2 -465.921} C_VEL
LIN {X 0,Y 608.5,Z 152.26,A -85,B 0,C 180,E1 -468.492,E2 -468.492} C_VEL
LIN {X 0,Y 608.566,Z 132.111,A -85,B 0,C 180,E1 -471.155,E2 -471.155} C_VEL
LIN {X 0,Y 608.442,Z 117.691,A -85,B 0,C 180,E1 -473.102,E2 -473.102} C_VEL
LIN {X 0,Y 608.476,Z 117.689,A -85,B 0,C 180,E1 -475.721,E2 -475.721} C_VEL
LIN {X 0,Y 608.454,Z 117.689,A -85,B 0,C 180,E1 -478.616,E2 -478.616} C_VEL
LIN {X 0,Y 608.448,Z 117.69,A -85,B 0,C 180,E1 -481.318,E2 -481.318} C_VEL
LIN {X 0,Y 608.475,Z 117.694,A -85,B 0,C 180,E1 -483.735,E2 -483.735} C_VEL
LIN {X 0,Y 608.442,Z 117.694,A -85,B 0,C 180,E1 -486.093,E2 -486.093} C_VEL
LIN {X 0,Y 608.427,Z 117.691,A -85,B 0,C 180,E1 -488.591,E2 -488.591} C_VEL
LIN {X 0,Y 608.467,Z 117.692,A -85,B 0,C 180,E1 -491.343,E2 -491.343} C_VEL
LIN {X 0,Y 608.447,Z 117.693,A -85,B 0,C 180,E1 -493.872,E2 -493.872} C_VEL
LIN {X 0,Y 608.464,Z 117.687,A -85,B 0,C 180,E1 -496.692,E2 -496.692} C_VEL
LIN {X 0,Y 608.438,Z 117.693,A -85,B 0,C 180,E1 -499.695,E2 -499.695} C_VEL
LIN {X 0,Y 608.48,Z 117.689,A -85,B 0,C 180,E1 -502.84,E2 -502.84} C_VEL
LIN {X 0,Y 608.449,Z 117.692,A -85,B 0,C 180,E1 -505.529,E2 -505.529} C_VEL
LIN {X 0,Y 608.427,Z 117.691,A -85,B 0,C 180,E1 -507.903,E2 -507.903} C_VEL
LIN {X 0,Y 608.435,Z 117.691,A -85,B 0,C 180,E1 -510.219,E2 -510.219} C_VEL
LIN {X 0,Y 608.48,Z 117.694,A -85,B 0,C 180,E1 -512.792,E2 -512.792} C_VEL
LIN {X 0,Y 608.419,Z 117.693,A -85,B 0,C 180,E1 -515.427,E2 -515.427} C_VEL
LIN {X 0,Y 608.456,Z 117.692,A -85,B 0,C 180,E1 -518.308,E2 -518.308} C_VEL
LIN {X 0,Y 608.411,Z 117.694,A -85,B 0,C 180,E1 -521.3,E2 -521.3} C_VEL
LIN {X 0,Y 608.424,Z 117.693,A -85,B 0,C 180,E1 -523.905,E2 -523.905} C_VEL
LIN {X 0,Y 608.429,Z 117.696,A -85,B 0,C 180,E1 -526.643,E2 -526.643} C_VEL
LIN {X 0,Y 608.4,Z 117.694,A -85,B 0,C 180,E1 -529.349,E2 -529.349} C_VEL
LIN {X 0,Y 608.431,Z 117.698,A -85,B 0,C 180,E1 -532.032,E2 -532.032} C_VEL
LIN {X 0,Y 608.412,Z 117.694,A -85,B 0,C 180,E1 -534.698,E2 -534.698} C_VEL
LIN {X 0,Y 608.425,Z 117.692,A -85,B 0,C 180,E1 -537.352,E2 -537.352} C_VEL
LIN {X 0,Y 608.473,Z 117.694,A -85,B 0,C 180,E1 -540,E2 -540} C_VEL
LIN {X 0,Y 608.425,Z 117.691,A -85,B 0,C 180,E1 -542.648,E2 -542.648} C_VEL
LIN {X 0,Y 608.429,Z 117.694,A -85,B 0,C 180,E1 -545.302,E2 -545.302} C_VEL
LIN {X 0,Y 608.468,Z 117.69,A -85,B 0,C 180,E1 -547.967,E2 -547.967} C_VEL
LIN {X 0,Y 608.439,Z 117.694,A -85,B 0,C 180,E1 -549.416,E2 -549.416} C_VEL
LIN {X 0,Y 607.77,Z 117.777,A -85,B 0,C 180,E1 -549.968,E2 -549.968} C_VEL
LIN {X 0,Y 604.927,Z 118.128,A -85,B 0,C 180,E1 -550.865,E2 -550.865} C_VEL
LIN {X 0,Y 602.518,Z 118.436,A -85,B 0,C 180,E1 -551.586,E2 -551.586} C_VEL
LIN {X 0,Y 601.471,Z 118.559,A -85,B 0,C 180,E1 -552.143,E2 -552.143} C_VEL
LIN {X 0,Y 601.378,Z 118.569,A -85,B 0,C 180,E1 -552.331,E2 -552.331} C_VEL
LIN {X 0,Y 601.384,Z 118.571,A -85,B 0,C 180,E1 -554.898,E2 -554.898} C_VEL
LIN {X 0,Y 601.385,Z 118.572,A -85,B 0,C 180,E1 -557.689,E2 -557.689} C_VEL
LIN {X 0,Y 601.39,Z 118.569,A -85,B 0,C 180,E1 -559.81,E2 -559.81} C_VEL
LIN {X 0,Y 601.401,Z 118.57,A -85,B 0,C 180,E1 -562.684,E2 -562.684} C_VEL
LIN {X 0,Y 601.425,Z 118.565,A -85,B 0,C 180,E1 -565.618,E2 -565.618} C_VEL
LIN {X 0,Y 601.387,Z 118.568,A -85,B 0,C 180,E1 -567.869,E2 -567.869} C_VEL
LIN {X 0,Y 601.399,Z 118.567,A -85,B 0,C 180,E1 -570.166,E2 -570.166} C_VEL
LIN {X 0,Y 601.412,Z 118.574,A -85,B 0,C 180,E1 -572.714,E2 -572.714} C_VEL
LIN {X 0,Y 601.397,Z 118.57,A -85,B 0,C 180,E1 -575.112,E2 -575.112} C_VEL
LIN {X 0,Y 601.434,Z 118.562,A -85,B 0,C 180,E1 -577.419,E2 -577.419} C_VEL
LIN {X 0,Y 601.401,Z 118.568,A -85,B 0,C 180,E1 -579.996,E2 -579.996} C_VEL
LIN {X 0,Y 601.414,Z 118.571,A -85,B 0,C 180,E1 -582.67,E2 -582.67} C_VEL
LIN {X 0,Y 601.401,Z 118.566,A -85,B 0,C 180,E1 -585.48,E2 -585.48} C_VEL
LIN {X 0,Y 601.424,Z 118.571,A -85,B 0,C 180,E1 -588.407,E2 -588.407} C_VEL
LIN {X 0,Y 601.433,Z 118.563,A -85,B 0,C 180,E1 -590.875,E2 -590.875} C_VEL
LIN {X 0,Y 601.4,Z 118.568,A -85,B 0,C 180,E1 -593.417,E2 -593.417} C_VEL
LIN {X 0,Y 601.434,Z 118.571,A -85,B 0,C 180,E1 -596.065,E2 -596.065} C_VEL
LIN {X 0,Y 601.422,Z 118.565,A -85,B 0,C 180,E1 -598.546,E2 -598.546} C_VEL
LIN {X 0,Y 601.424,Z 118.567,A -85,B 0,C 180,E1 -601.373,E2 -601.373} C_VEL
LIN {X 0,Y 601.401,Z 118.576,A -85,B 0,C 180,E1 -603.636,E2 -603.636} C_VEL
LIN {X 0,Y 601.426,Z 118.564,A -85,B 0,C 180,E1 -606.59,E2 -606.59} C_VEL
LIN {X 0,Y 601.43,Z 118.626,A -85,B 0,C 180,E1 -606.909,E2 -606.909} C_VEL
LIN {X 0,Y 601.424,Z 132.995,A -85,B 0,C 180,E1 -609.478,E2 -609.478} C_VEL
LIN {X 0,Y 601.376,Z 146.611,A -85,B 0,C 180,E1 -611.882,E2 -611.882} C_VEL
LIN {X 0,Y 601.661,Z 150.731,A -85,B 0,C 180,E1 -611.946,E2 -611.946} C_VEL
LIN {X 0,Y 601.551,Z 253.342,A -85,B 0,C 180,E1 -613.191,E2 -613.191} C_VEL
LIN {X 0,Y 601.535,Z 266.804,A -85,B 0,C 180,E1 -613.499,E2 -613.499} C_VEL
LIN {X 0,Y 601.539,Z 279.56,A -85,B 0,C 180,E1 -613.933,E2 -613.933} C_VEL
LIN {X 0,Y 601.471,Z 291.683,A -85,B 0,C 180,E1 -614.497,E2 -614.497} C_VEL
LIN {X 0,Y 601.462,Z 303.247,A -85,B 0,C 180,E1 -615.19,E2 -615.19} C_VEL
LIN {X 0,Y 601.444,Z 312.815,A -85,B 0,C 180,E1 -615.901,E2 -615.901} C_VEL
LIN {X 0,Y 601.445,Z 321.221,A -85,B 0,C 180,E1 -616.656,E2 -616.656} C_VEL
LIN {X 0,Y 601.398,Z 329.158,A -85,B 0,C 180,E1 -617.514,E2 -617.514} C_VEL
LIN {X 0,Y 601.391,Z 336.872,A -85,B 0,C 180,E1 -618.541,E2 -618.541} C_VEL
LIN {X 0,Y 601.371,Z 343.048,A -85,B 0,C 180,E1 -619.563,E2 -619.563} C_VEL
LIN {X 0,Y 601.345,Z 347.923,A -85,B 0,C 180,E1 -620.582,E2 -620.582} C_VEL
LIN {X 0,Y 601.35,Z 351.655,A -85,B 0,C 180,E1 -621.599,E2 -621.599} C_VEL
LIN {X 0,Y 601.323,Z 354.353,A -85,B 0,C 180,E1 -622.613,E2 -622.613} C_VEL
LIN {X 0,Y 601.349,Z 355.827,A -85,B 0,C 180,E1 -623.416,E2 -623.416} C_VEL
LIN {X 0,Y 601.336,Z 356.911,A -85,B 0,C 180,E1 -624.635,E2 -624.635} C_VEL
LIN {X 0,Y 601.343,Z 356.601,A -85,B 0,C 180,E1 -625.978,E2 -625.978} C_VEL
LIN {X 0,Y 601.338,Z 355.863,A -85,B 0,C 180,E1 -626.649,E2 -626.649} C_VEL
LIN {X 0,Y 601.344,Z 353.11,A -85,B 0,C 180,E1 -627.99,E2 -627.99} C_VEL
LIN {X 0,Y 601.335,Z 349.939,A -85,B 0,C 180,E1 -628.995,E2 -628.995} C_VEL
LIN {X 0,Y 601.358,Z 345.721,A -85,B 0,C 180,E1 -629.999,E2 -629.999} C_VEL
LIN {X 0,Y 601.387,Z 339.333,A -85,B 0,C 180,E1 -631.171,E2 -631.171} C_VEL
LIN {X 0,Y 601.384,Z 332.379,A -85,B 0,C 180,E1 -632.176,E2 -632.176} C_VEL
LIN {X 0,Y 601.395,Z 323.692,A -85,B 0,C 180,E1 -633.181,E2 -633.181} C_VEL
LIN {X 0,Y 601.447,Z 313.857,A -85,B 0,C 180,E1 -634.104,E2 -634.104} C_VEL
LIN {X 0,Y 601.451,Z 303.864,A -85,B 0,C 180,E1 -634.859,E2 -634.859} C_VEL
LIN {X 0,Y 601.487,Z 292.824,A -85,B 0,C 180,E1 -635.531,E2 -635.531} C_VEL
LIN {X 0,Y 601.546,Z 280.272,A -85,B 0,C 180,E1 -636.128,E2 -636.128} C_VEL
LIN {X 0,Y 601.528,Z 267.667,A -85,B 0,C 180,E1 -636.567,E2 -636.567} C_VEL
LIN {X 0,Y 601.551,Z 254.01,A -85,B 0,C 180,E1 -636.887,E2 -636.887} C_VEL
LIN {X 0,Y 601.62,Z 207.331,A -85,B 0,C 180,E1 -637.467,E2 -637.467} C_VEL
LIN {X 0,Y 601.509,Z 147.544,A -85,B 0,C 180,E1 -638.186,E2 -638.186} C_VEL
LIN {X 0,Y 601.398,Z 146.606,A -85,B 0,C 180,E1 -638.209,E2 -638.209} C_VEL
LIN {X 0,Y 601.436,Z 130.728,A -85,B 0,C 180,E1 -641.015,E2 -641.015} C_VEL
LIN {X 0,Y 601.399,Z 118.569,A -85,B 0,C 180,E1 -643.214,E2 -643.214} C_VEL
LIN {X 0,Y 601.408,Z 118.566,A -85,B 0,C 180,E1 -645.591,E2 -645.591} C_VEL
LIN {X 0,Y 601.416,Z 118.574,A -85,B 0,C 180,E1 -648.391,E2 -648.391} C_VEL
LIN {X 0,Y 601.405,Z 118.566,A -85,B 0,C 180,E1 -651.238,E2 -651.238} C_VEL
LIN {X 0,Y 601.461,Z 118.569,A -85,B 0,C 180,E1 -654.139,E2 -654.139} C_VEL
LIN {X 0,Y 601.44,Z 118.561,A -85,B 0,C 180,E1 -657.111,E2 -657.111} C_VEL
LIN {X 0,Y 601.425,Z 118.57,A -85,B 0,C 180,E1 -660.163,E2 -660.163} C_VEL
LIN {X 0,Y 601.405,Z 118.566,A -85,B 0,C 180,E1 -662.712,E2 -662.712} C_VEL
LIN {X 0,Y 601.388,Z 118.569,A -85,B 0,C 180,E1 -665.11,E2 -665.11} C_VEL
LIN {X 0,Y 601.432,Z 118.568,A -85,B 0,C 180,E1 -667.418,E2 -667.418} C_VEL
LIN {X 0,Y 601.407,Z 118.57,A -85,B 0,C 180,E1 -669.994,E2 -669.994} C_VEL
LIN {X 0,Y 601.4,Z 118.567,A -85,B 0,C 180,E1 -672.67,E2 -672.67} C_VEL
LIN {X 0,Y 601.42,Z 118.574,A -85,B 0,C 180,E1 -675.481,E2 -675.481} C_VEL
LIN {X 0,Y 601.408,Z 118.566,A -85,B 0,C 180,E1 -678.407,E2 -678.407} C_VEL
LIN {X 0,Y 601.403,Z 118.57,A -85,B 0,C 180,E1 -680.872,E2 -680.872} C_VEL
LIN {X 0,Y 601.397,Z 118.573,A -85,B 0,C 180,E1 -683.416,E2 -683.416} C_VEL
LIN {X 0,Y 601.405,Z 118.566,A -85,B 0,C 180,E1 -686.066,E2 -686.066} C_VEL
LIN {X 0,Y 601.417,Z 118.567,A -85,B 0,C 180,E1 -688.543,E2 -688.543} C_VEL
LIN {X 0,Y 601.399,Z 118.57,A -85,B 0,C 180,E1 -691.371,E2 -691.371} C_VEL
LIN {X 0,Y 601.377,Z 118.57,A -85,B 0,C 180,E1 -693.635,E2 -693.635} C_VEL
LIN {X 0,Y 601.394,Z 118.567,A -85,B 0,C 180,E1 -695.857,E2 -695.857} C_VEL
LIN {X 0,Y 601.389,Z 118.577,A -85,B 0,C 180,E1 -698.76,E2 -698.76} C_VEL
LIN {X 0,Y 601.357,Z 118.572,A -85,B 0,C 180,E1 -701.606,E2 -701.606} C_VEL
LIN {X 0,Y 601.388,Z 118.577,A -85,B 0,C 180,E1 -704.408,E2 -704.408} C_VEL
LIN {X 0,Y 601.353,Z 118.573,A -85,B 0,C 180,E1 -707.17,E2 -707.17} C_VEL
LIN {X 0,Y 601.414,Z 118.569,A -85,B 0,C 180,E1 -709.905,E2 -709.905} C_VEL
LIN {X 0,Y 601.381,Z 118.573,A -85,B 0,C 180,E1 -712.614,E2 -712.614} C_VEL
LIN {X 0,Y 601.387,Z 118.571,A -85,B 0,C 180,E1 -714.635,E2 -714.635} C_VEL
LIN {X 0,Y 601.385,Z 118.569,A -85,B 0,C 180,E1 -717.321,E2 -717.321} C_VEL
LIN {X 0,Y 601.433,Z 118.572,A -85,B 0,C 180,E1 -720,E2 -720} C_VEL
LIN {X 0,Y 601.387,Z 118.569,A -85,B 0,C 180,E1 -722.679,E2 -722.679} C_VEL
LIN {X 0,Y 601.391,Z 118.571,A -85,B 0,C 180,E1 -725.364,E2 -725.364} C_VEL
LIN {X 0,Y 601.422,Z 118.568,A -85,B 0,C 180,E1 -728.061,E2 -728.061} C_VEL
LIN {X 0,Y 601.386,Z 118.57,A -85,B 0,C 180,E1 -731,E2 -731} C_VEL
LIN {X 0,Y 601.391,Z 118.578,A -85,B 0,C 180,E1 -733.516,E2 -733.516} C_VEL
LIN {X 0,Y 601.389,Z 118.568,A -85,B 0,C 180,E1 -736.288,E2 -736.288} C_VEL
LIN {X 0,Y 601.398,Z 118.573,A -85,B 0,C 180,E1 -739.1,E2 -739.1} C_VEL
LIN {X 0,Y 601.387,Z 118.569,A -85,B 0,C 180,E1 -741.96,E2 -741.96} C_VEL
LIN {X 0,Y 601.384,Z 118.574,A -85,B 0,C 180,E1 -744.879,E2 -744.879} C_VEL
LIN {X 0,Y 601.412,Z 118.571,A -85,B 0,C 180,E1 -747.365,E2 -747.365} C_VEL
LIN {X 0,Y 601.388,Z 118.568,A -85,B 0,C 180,E1 -750.166,E2 -750.166} C_VEL
LIN {X 0,Y 601.4,Z 118.573,A -85,B 0,C 180,E1 -752.715,E2 -752.715} C_VEL
LIN {X 0,Y 601.393,Z 118.573,A -85,B 0,C 180,E1 -755.114,E2 -755.114} C_VEL
LIN {X 0,Y 601.426,Z 118.564,A -85,B 0,C 180,E1 -757.42,E2 -757.42} C_VEL
LIN {X 0,Y 601.392,Z 118.569,A -85,B 0,C 180,E1 -759.997,E2 -759.997} C_VEL
LIN {X 0,Y 601.405,Z 118.575,A -85,B 0,C 180,E1 -762.671,E2 -762.671} C_VEL
LIN {X 0,Y 601.391,Z 118.568,A -85,B 0,C 180,E1 -765.48,E2 -765.48} C_VEL
LIN {X 0,Y 601.419,Z 118.574,A -85,B 0,C 180,E1 -768.408,E2 -768.408} C_VEL
LIN {X 0,Y 601.428,Z 118.565,A -85,B 0,C 180,E1 -770.876,E2 -770.876} C_VEL
LIN {X 0,Y 601.394,Z 118.567,A -85,B 0,C 180,E1 -773.418,E2 -773.418} C_VEL
LIN {X 0,Y 601.429,Z 118.572,A -85,B 0,C 180,E1 -776.065,E2 -776.065} C_VEL
LIN {X 0,Y 601.424,Z 118.563,A -85,B 0,C 180,E1 -779.059,E2 -779.059} C_VEL
LIN {X 0,Y 601.413,Z 118.567,A -85,B 0,C 180,E1 -781.373,E2 -781.373} C_VEL
LIN {X 0,Y 601.394,Z 118.573,A -85,B 0,C 180,E1 -783.637,E2 -783.637} C_VEL
LIN {X 0,Y 601.421,Z 118.568,A -85,B 0,C 180,E1 -786.591,E2 -786.591} C_VEL
LIN {X 0,Y 601.448,Z 118.824,A -85,B 0,C 180,E1 -786.774,E2 -786.774} C_VEL
LIN {X 0,Y 601.693,Z 125.513,A -85,B 0,C 180,E1 -787.697,E2 -787.697} C_VEL
LIN {X 0,Y 601.616,Z 146.746,A -85,B 0,C 180,E1 -790.554,E2 -790.554} C_VEL
LIN {X 0,Y 601.511,Z 167.906,A -85,B 0,C 180,E1 -793.352,E2 -793.352} C_VEL
LIN {X 0,Y 601.466,Z 189.677,A -85,B 0,C 180,E1 -796.191,E2 -796.191} C_VEL
LIN {X 0,Y 601.425,Z 194.528,A -85,B 0,C 180,E1 -796.818,E2 -796.818} C_VEL
LIN {X 0,Y 601.625,Z 214.886,A -85,B 0,C 180,E1 -797.07,E2 -797.07} C_VEL
LIN {X 0,Y 601.613,Z 302.989,A -85,B 0,C 180,E1 -798.14,E2 -798.14} C_VEL
LIN {X 0,Y 601.559,Z 316.246,A -85,B 0,C 180,E1 -798.438,E2 -798.438} C_VEL
LIN {X 0,Y 601.542,Z 328.646,A -85,B 0,C 180,E1 -798.853,E2 -798.853} C_VEL
LIN {X 0,Y 601.522,Z 340.648,A -85,B 0,C 180,E1 -799.397,E2 -799.397} C_VEL
LIN {X 0,Y 601.483,Z 352.211,A -85,B 0,C 180,E1 -800.077,E2 -800.077} C_VEL
LIN {X 0,Y 601.444,Z 362.605,A -85,B 0,C 180,E1 -800.84,E2 -800.84} C_VEL
LIN {X 0,Y 601.429,Z 371.12,A -85,B 0,C 180,E1 -801.602,E2 -801.602} C_VEL
LIN {X 0,Y 601.417,Z 378.967,A -85,B 0,C 180,E1 -802.447,E2 -802.447} C_VEL
LIN {X 0,Y 601.369,Z 386.228,A -85,B 0,C 180,E1 -803.398,E2 -803.398} C_VEL
LIN {X 0,Y 601.372,Z 391.87,A -85,B 0,C 180,E1 -804.3,E2 -804.3} C_VEL
LIN {X 0,Y 601.336,Z 396.953,A -85,B 0,C 180,E1 -805.308,E2 -805.308} C_VEL
LIN {X 0,Y 601.368,Z 400.898,A -85,B 0,C 180,E1 -806.315,E2 -806.315} C_VEL
LIN {X 0,Y 601.325,Z 403.811,A -85,B 0,C 180,E1 -807.321,E2 -807.321} C_VEL
LIN {X 0,Y 601.343,Z 405.203,A -85,B 0,C 180,E1 -807.991,E2 -807.991} C_VEL
LIN {X 0,Y 601.339,Z 406.784,A -85,B 0,C 180,E1 -809.331,E2 -809.331} C_VEL
LIN {X 0,Y 601.335,Z 407,A -85,B 0,C 180,E1 -810.001,E2 -810.001} C_VEL
LIN {X 0,Y 601.347,Z 406.184,A -85,B 0,C 180,E1 -811.34,E2 -811.34} C_VEL
LIN {X 0,Y 601.343,Z 405.201,A -85,B 0,C 180,E1 -812.01,E2 -812.01} C_VEL
LIN {X 0,Y 601.325,Z 403.808,A -85,B 0,C 180,E1 -812.68,E2 -812.68} C_VEL
LIN {X 0,Y 601.368,Z 400.894,A -85,B 0,C 180,E1 -813.686,E2 -813.686} C_VEL
LIN {X 0,Y 601.336,Z 396.947,A -85,B 0,C 180,E1 -814.693,E2 -814.693} C_VEL
LIN {X 0,Y 601.373,Z 390.874,A -85,B 0,C 180,E1 -815.87,E2 -815.87} C_VEL
LIN {X 0,Y 601.382,Z 384.232,A -85,B 0,C 180,E1 -816.88,E2 -816.88} C_VEL
LIN {X 0,Y 601.401,Z 375.985,A -85,B 0,C 180,E1 -817.893,E2 -817.893} C_VEL
LIN {X 0,Y 601.436,Z 367.531,A -85,B 0,C 180,E1 -818.738,E2 -818.738} C_VEL
LIN {X 0,Y 601.449,Z 357.086,A -85,B 0,C 180,E1 -819.586,E2 -819.586} C_VEL
LIN {X 0,Y 601.467,Z 346.75,A -85,B 0,C 180,E1 -820.265,E2 -820.265} C_VEL
LIN {X 0,Y 601.538,Z 334.593,A -85,B 0,C 180,E1 -820.896,E2 -820.896} C_VEL
LIN {X 0,Y 601.555,Z 322.205,A -85,B 0,C 180,E1 -821.379,E2 -821.379} C_VEL
LIN {X 0,Y 601.583,Z 309.418,A -85,B 0,C 180,E1 -821.733,E2 -821.733} C_VEL
LIN {X 0,Y 601.619,Z 297.049,A -85,B 0,C 180,E1 -821.946,E2 -821.946} C_VEL
LIN {X 0,Y 601.489,Z 195.105,A -85,B 0,C 180,E1 -823.171,E2 -823.171} C_VEL
LIN {X 0,Y 601.444,Z 194.269,A -85,B 0,C 180,E1 -823.215,E2 -823.215} C_VEL
LIN {X 0,Y 601.516,Z 171.998,A -85,B 0,C 180,E1 -826.111,E2 -826.111} C_VEL
LIN {X 0,Y 601.532,Z 152.091,A -85,B 0,C 180,E1 -828.737,E2 -828.737} C_VEL
LIN {X 0,Y 601.656,Z 132.111,A -85,B 0,C 180,E1 -831.41,E2 -831.41} C_VEL
LIN {X 0,Y 601.673,Z 120.144,A -85,B 0,C 180,E1 -833.036,E2 -833.036} C_VEL
LIN {X 0,Y 601.409,Z 118.569,A -85,B 0,C 180,E1 -833.274,E2 -833.274} C_VEL
LIN {X 0,Y 601.413,Z 118.571,A -85,B 0,C 180,E1 -835.867,E2 -835.867} C_VEL
LIN {X 0,Y 601.417,Z 118.565,A -85,B 0,C 180,E1 -838.785,E2 -838.785} C_VEL
LIN {X 0,Y 601.398,Z 118.574,A -85,B 0,C 180,E1 -841.727,E2 -841.727} C_VEL
LIN {X 0,Y 601.423,Z 118.569,A -85,B 0,C 180,E1 -844.119,E2 -844.119} C_VEL
LIN {X 0,Y 601.396,Z 118.567,A -85,B 0,C 180,E1 -846.584,E2 -846.584} C_VEL
LIN {X 0,Y 601.44,Z 118.57,A -85,B 0,C 180,E1 -849.535,E2 -849.535} C_VEL
LIN {X 0,Y 601.413,Z 118.571,A -85,B 0,C 180,E1 -851.766,E2 -851.766} C_VEL
LIN {X 0,Y 601.399,Z 118.567,A -85,B 0,C 180,E1 -854.532,E2 -854.532} C_VEL
LIN {X 0,Y 601.406,Z 118.575,A -85,B 0,C 180,E1 -857.41,E2 -857.41} C_VEL
LIN {X 0,Y 601.389,Z 118.569,A -85,B 0,C 180,E1 -860.003,E2 -860.003} C_VEL
LIN {X 0,Y 601.434,Z 118.564,A -85,B 0,C 180,E1 -862.618,E2 -862.618} C_VEL
LIN {X 0,Y 601.404,Z 118.566,A -85,B 0,C 180,E1 -865.88,E2 -865.88} C_VEL
LIN {X 0,Y 601.413,Z 118.568,A -85,B 0,C 180,E1 -868.546,E2 -868.546} C_VEL
LIN {X 0,Y 601.395,Z 118.57,A -85,B 0,C 180,E1 -871.371,E2 -871.371} C_VEL
LIN {X 0,Y 601.377,Z 118.569,A -85,B 0,C 180,E1 -873.635,E2 -873.635} C_VEL
LIN {X 0,Y 601.394,Z 118.567,A -85,B 0,C 180,E1 -875.857,E2 -875.857} C_VEL
LIN {X 0,Y 601.391,Z 118.575,A -85,B 0,C 180,E1 -878.76,E2 -878.76} C_VEL
LIN {X 0,Y 601.357,Z 118.572,A -85,B 0,C 180,E1 -881.606,E2 -881.606} C_VEL
LIN {X 0,Y 601.385,Z 118.578,A -85,B 0,C 180,E1 -884.408,E2 -884.408} C_VEL
LIN {X 0,Y 601.384,Z 118.576,A -85,B 0,C 180,E1 -886.483,E2 -886.483} C_VEL
LIN {X 0,Y 601.348,Z 118.573,A -85,B 0,C 180,E1 -889.223,E2 -889.223} C_VEL
LIN {X 0,Y 601.399,Z 118.572,A -85,B 0,C 180,E1 -891.939,E2 -891.939} C_VEL
LIN {X 0,Y 601.384,Z 118.571,A -85,B 0,C 180,E1 -894.636,E2 -894.636} C_VEL
LIN {X 0,Y 601.393,Z 118.568,A -85,B 0,C 180,E1 -897.321,E2 -897.321} C_VEL
LIN {X 0,Y 601.441,Z 118.57,A -85,B 0,C 180,E1 -900,E2 -900} C_VEL
LIN {X 0,Y 601.394,Z 118.567,A -85,B 0,C 180,E1 -902.679,E2 -902.679} C_VEL
LIN {X 0,Y 601.398,Z 118.571,A -85,B 0,C 180,E1 -905.364,E2 -905.364} C_VEL
LIN {X 0,Y 601.428,Z 118.566,A -85,B 0,C 180,E1 -908.061,E2 -908.061} C_VEL
LIN {X 0,Y 601.396,Z 118.569,A -85,B 0,C 180,E1 -910.999,E2 -910.999} C_VEL
LIN {X 0,Y 601.378,Z 118.569,A -85,B 0,C 180,E1 -912.331,E2 -912.331} C_VEL
LIN {X 0,Y 600.693,Z 118.657,A -85,B 0,C 180,E1 -912.891,E2 -912.891} C_VEL
LIN {X 0,Y 597.842,Z 119.013,A -85,B 0,C 180,E1 -913.799,E2 -913.799} C_VEL
LIN {X 0,Y 595.445,Z 119.313,A -85,B 0,C 180,E1 -914.529,E2 -914.529} C_VEL
LIN {X 0,Y 594.416,Z 119.441,A -85,B 0,C 180,E1 -915.092,E2 -915.092} C_VEL
LIN {X 0,Y 594.332,Z 119.45,A -85,B 0,C 180,E1 -915.283,E2 -915.283} C_VEL
LIN {X 0,Y 594.331,Z 119.448,A -85,B 0,C 180,E1 -917.906,E2 -917.906} C_VEL
LIN {X 0,Y 594.381,Z 119.444,A -85,B 0,C 180,E1 -920.777,E2 -920.777} C_VEL
LIN {X 0,Y 594.35,Z 119.446,A -85,B 0,C 180,E1 -923.706,E2 -923.706} C_VEL
LIN {X 0,Y 594.351,Z 119.444,A -85,B 0,C 180,E1 -926.016,E2 -926.016} C_VEL
LIN {X 0,Y 594.362,Z 119.444,A -85,B 0,C 180,E1 -928.228,E2 -928.228} C_VEL
LIN {X 0,Y 594.366,Z 119.448,A -85,B 0,C 180,E1 -930.561,E2 -930.561} C_VEL
LIN {X 0,Y 594.376,Z 119.448,A -85,B 0,C 180,E1 -932.951,E2 -932.951} C_VEL
LIN {X 0,Y 594.349,Z 119.445,A -85,B 0,C 180,E1 -935.409,E2 -935.409} C_VEL
LIN {X 0,Y 594.376,Z 119.443,A -85,B 0,C 180,E1 -937.942,E2 -937.942} C_VEL
LIN {X 0,Y 594.375,Z 119.445,A -85,B 0,C 180,E1 -940.822,E2 -940.822} C_VEL
LIN {X 0,Y 594.355,Z 119.444,A -85,B 0,C 180,E1 -943.301,E2 -943.301} C_VEL
LIN {X 0,Y 594.363,Z 119.45,A -85,B 0,C 180,E1 -946.161,E2 -946.161} C_VEL
LIN {X 0,Y 594.375,Z 119.442,A -85,B 0,C 180,E1 -949.179,E2 -949.179} C_VEL
LIN {X 0,Y 594.384,Z 119.45,A -85,B 0,C 180,E1 -952.059,E2 -952.059} C_VEL
LIN {X 0,Y 594.352,Z 119.446,A -85,B 0,C 180,E1 -954.677,E2 -954.677} C_VEL
LIN {X 0,Y 594.38,Z 119.441,A -85,B 0,C 180,E1 -957.089,E2 -957.089} C_VEL
LIN {X 0,Y 594.39,Z 119.447,A -85,B 0,C 180,E1 -959.672,E2 -959.672} C_VEL
LIN {X 0,Y 594.38,Z 119.442,A -85,B 0,C 180,E1 -962.539,E2 -962.539} C_VEL
LIN {X 0,Y 594.375,Z 119.442,A -85,B 0,C 180,E1 -964.807,E2 -964.807} C_VEL
LIN {X 0,Y 594.385,Z 119.521,A -85,B 0,C 180,E1 -966.849,E2 -966.849} C_VEL
LIN {X 0,Y 594.408,Z 132.634,A -85,B 0,C 180,E1 -969.224,E2 -969.224} C_VEL
LIN {X 0,Y 594.33,Z 146.631,A -85,B 0,C 180,E1 -971.726,E2 -971.726} C_VEL
LIN {X 0,Y 594.747,Z 151.111,A -85,B 0,C 180,E1 -971.795,E2 -971.795} C_VEL
LIN {X 0,Y 594.603,Z 253.415,A -85,B 0,C 180,E1 -973.052,E2 -973.052} C_VEL
LIN {X 0,Y 594.564,Z 266.636,A -85,B 0,C 180,E1 -973.357,E2 -973.357} C_VEL
LIN {X 0,Y 594.581,Z 279.112,A -85,B 0,C 180,E1 -973.784,E2 -973.784} C_VEL
LIN {X 0,Y 594.512,Z 290.557,A -85,B 0,C 180,E1 -974.311,E2 -974.311} C_VEL
LIN {X 0,Y 594.455,Z 302.338,A -85,B 0,C 180,E1 -975.011,E2 -975.011} C_VEL
LIN {X 0,Y 594.426,Z 313.082,A -85,B 0,C 180,E1 -975.814,E2 -975.814} C_VEL
LIN {X 0,Y 594.396,Z 322.335,A -85,B 0,C 180,E1 -976.669,E2 -976.669} C_VEL
LIN {X 0,Y 594.349,Z 331.44,A -85,B 0,C 180,E1 -977.71,E2 -977.71} C_VEL
LIN {X 0,Y 594.323,Z 338.743,A -85,B 0,C 180,E1 -978.748,E2 -978.748} C_VEL
LIN {X 0,Y 594.261,Z 344.535,A -85,B 0,C 180,E1 -979.781,E2 -979.781} C_VEL
LIN {X 0,Y 594.262,Z 349.081,A -85,B 0,C 180,E1 -980.813,E2 -980.813} C_VEL
LIN {X 0,Y 594.272,Z 352.522,A -85,B 0,C 180,E1 -981.841,E2 -981.841} C_VEL
LIN {X 0,Y 594.249,Z 354.228,A -85,B 0,C 180,E1 -982.524,E2 -982.524} C_VEL
LIN {X 0,Y 594.264,Z 355.869,A -85,B 0,C 180,E1 -983.425,E2 -983.425} C_VEL
LIN {X 0,Y 594.252,Z 356.897,A -85,B 0,C 180,E1 -984.57,E2 -984.57} C_VEL
LIN {X 0,Y 594.256,Z 356.642,A -85,B 0,C 180,E1 -985.93,E2 -985.93} C_VEL
LIN {X 0,Y 594.258,Z 355.941,A -85,B 0,C 180,E1 -986.609,E2 -986.609} C_VEL
LIN {X 0,Y 594.223,Z 354.814,A -85,B 0,C 180,E1 -987.288,E2 -987.288} C_VEL
LIN {X 0,Y 594.243,Z 353.265,A -85,B 0,C 180,E1 -987.966,E2 -987.966} C_VEL
LIN {X 0,Y 594.248,Z 350.154,A -85,B 0,C 180,E1 -988.983,E2 -988.983} C_VEL
LIN {X 0,Y 594.283,Z 346.002,A -85,B 0,C 180,E1 -989.999,E2 -989.999} C_VEL
LIN {X 0,Y 594.325,Z 339.685,A -85,B 0,C 180,E1 -991.185,E2 -991.185} C_VEL
LIN {X 0,Y 594.319,Z 332.824,A -85,B 0,C 180,E1 -992.202,E2 -992.202} C_VEL
LIN {X 0,Y 594.334,Z 324.257,A -85,B 0,C 180,E1 -993.219,E2 -993.219} C_VEL
LIN {X 0,Y 594.373,Z 315.5,A -85,B 0,C 180,E1 -994.068,E2 -994.068} C_VEL
LIN {X 0,Y 594.425,Z 304.743,A -85,B 0,C 180,E1 -994.917,E2 -994.917} C_VEL
LIN {X 0,Y 594.5,Z 293.908,A -85,B 0,C 180,E1 -995.596,E2 -995.596} C_VEL
LIN {X 0,Y 594.585,Z 281.521,A -85,B 0,C 180,E1 -996.205,E2 -996.205} C_VEL
LIN {X 0,Y 594.563,Z 269.336,A -85,B 0,C 180,E1 -996.655,E2 -996.655} C_VEL
LIN {X 0,Y 594.604,Z 256.037,A -85,B 0,C 180,E1 -996.989,E2 -996.989} C_VEL
LIN {X 0,Y 594.662,Z 236.759,A -85,B 0,C 180,E1 -997.258,E2 -997.258} C_VEL
LIN {X 0,Y 594.706,Z 148.861,A -85,B 0,C 180,E1 -998.323,E2 -998.323} C_VEL
LIN {X 0,Y 594.368,Z 146.587,A -85,B 0,C 180,E1 -998.371,E2 -998.371} C_VEL
LIN {X 0,Y 594.442,Z 130.446,A -85,B 0,C 180,E1 -1001.259,E2 -1001.259} C_VEL
LIN {X 0,Y 594.367,Z 119.446,A -85,B 0,C 180,E1 -1003.287,E2 -1003.287} C_VEL
LIN {X 0,Y 594.364,Z 119.445,A -85,B 0,C 180,E1 -1005.78,E2 -1005.78} C_VEL
LIN {X 0,Y 594.379,Z 119.446,A -85,B 0,C 180,E1 -1008.617,E2 -1008.617} C_VEL
LIN {X 0,Y 594.365,Z 119.444,A -85,B 0,C 180,E1 -1011.502,E2 -1011.502} C_VEL
LIN {X 0,Y 594.389,Z 119.445,A -85,B 0,C 180,E1 -1014.445,E2 -1014.445} C_VEL
LIN {X 0,Y 594.375,Z 119.443,A -85,B 0,C 180,E1 -1016.699,E2 -1016.699} C_VEL
LIN {X 0,Y 594.373,Z 119.442,A -85,B 0,C 180,E1 -1018.998,E2 -1018.998} C_VEL
LIN {X 0,Y 594.38,Z 119.447,A -85,B 0,C 180,E1 -1021.642,E2 -1021.642} C_VEL
LIN {X 0,Y 594.37,Z 119.443,A -85,B 0,C 180,E1 -1024.579,E2 -1024.579} C_VEL
LIN {X 0,Y 594.384,Z 119.449,A -85,B 0,C 180,E1 -1027.607,E2 -1027.607} C_VEL
LIN {X 0,Y 594.356,Z 119.444,A -85,B 0,C 180,E1 -1030.567,E2 -1030.567} C_VEL
LIN {X 0,Y 594.36,Z 119.45,A -85,B 0,C 180,E1 -1033.298,E2 -1033.298} C_VEL
LIN {X 0,Y 594.344,Z 119.446,A -85,B 0,C 180,E1 -1036.161,E2 -1036.161} C_VEL
LIN {X 0,Y 594.367,Z 119.443,A -85,B 0,C 180,E1 -1038.535,E2 -1038.535} C_VEL
LIN {X 0,Y 594.364,Z 119.453,A -85,B 0,C 180,E1 -1041.296,E2 -1041.296} C_VEL
LIN {X 0,Y 594.337,Z 119.448,A -85,B 0,C 180,E1 -1043.754,E2 -1043.754} C_VEL
LIN {X 0,Y 594.353,Z 119.445,A -85,B 0,C 180,E1 -1046.237,E2 -1046.237} C_VEL
LIN {X 0,Y 594.363,Z 119.448,A -85,B 0,C 180,E1 -1048.649,E2 -1048.649} C_VEL
LIN {X 0,Y 594.367,Z 119.451,A -85,B 0,C 180,E1 -1051.042,E2 -1051.042} C_VEL
LIN {X 0,Y 594.37,Z 119.446,A -85,B 0,C 180,E1 -1053.3,E2 -1053.3} C_VEL
LIN {X 0,Y 594.331,Z 119.448,A -85,B 0,C 180,E1 -1055.575,E2 -1055.575} C_VEL
LIN {X 0,Y 594.347,Z 119.452,A -85,B 0,C 180,E1 -1058.496,E2 -1058.496} C_VEL
LIN {X 0,Y 594.337,Z 119.447,A -85,B 0,C 180,E1 -1061.381,E2 -1061.381} C_VEL
LIN {X 0,Y 594.341,Z 119.446,A -85,B 0,C 180,E1 -1063.513,E2 -1063.513} C_VEL
LIN {X 0,Y 594.352,Z 119.453,A -85,B 0,C 180,E1 -1066.32,E2 -1066.32} C_VEL
LIN {X 0,Y 594.331,Z 119.448,A -85,B 0,C 180,E1 -1069.094,E2 -1069.094} C_VEL
LIN {X 0,Y 594.362,Z 119.447,A -85,B 0,C 180,E1 -1071.842,E2 -1071.842} C_VEL
LIN {X 0,Y 594.358,Z 119.448,A -85,B 0,C 180,E1 -1074.572,E2 -1074.572} C_VEL
LIN {X 0,Y 594.353,Z 119.445,A -85,B 0,C 180,E1 -1077.289,E2 -1077.289} C_VEL
LIN {X 0,Y 594.401,Z 119.448,A -85,B 0,C 180,E1 -1080,E2 -1080} C_VEL
LIN {X 0,Y 594.355,Z 119.445,A -85,B 0,C 180,E1 -1082.711,E2 -1082.711} C_VEL
LIN {X 0,Y 594.361,Z 119.448,A -85,B 0,C 180,E1 -1085.428,E2 -1085.428} C_VEL
LIN {X 0,Y 594.364,Z 119.446,A -85,B 0,C 180,E1 -1088.157,E2 -1088.157} C_VEL
LIN {X 0,Y 594.352,Z 119.447,A -85,B 0,C 180,E1 -1091.062,E2 -1091.062} C_VEL
LIN {X 0,Y 594.354,Z 119.452,A -85,B 0,C 180,E1 -1093.68,E2 -1093.68} C_VEL
LIN {X 0,Y 594.34,Z 119.447,A -85,B 0,C 180,E1 -1096.706,E2 -1096.706} C_VEL
LIN {X 0,Y 594.349,Z 119.455,A -85,B 0,C 180,E1 -1099.335,E2 -1099.335} C_VEL
LIN {X 0,Y 594.347,Z 119.452,A -85,B 0,C 180,E1 -1101.504,E2 -1101.504} C_VEL
LIN {X 0,Y 594.331,Z 119.448,A -85,B 0,C 180,E1 -1104.449,E2 -1104.449} C_VEL
LIN {X 0,Y 594.372,Z 119.446,A -85,B 0,C 180,E1 -1106.7,E2 -1106.7} C_VEL
LIN {X 0,Y 594.366,Z 119.453,A -85,B 0,C 180,E1 -1108.999,E2 -1108.999} C_VEL
LIN {X 0,Y 594.376,Z 119.443,A -85,B 0,C 180,E1 -1111.645,E2 -1111.645} C_VEL
LIN {X 0,Y 594.373,Z 119.448,A -85,B 0,C 180,E1 -1114.581,E2 -1114.581} C_VEL
LIN {X 0,Y 594.378,Z 119.442,A -85,B 0,C 180,E1 -1117.609,E2 -1117.609} C_VEL
LIN {X 0,Y 594.355,Z 119.453,A -85,B 0,C 180,E1 -1120.568,E2 -1120.568} C_VEL
LIN {X 0,Y 594.358,Z 119.444,A -85,B 0,C 180,E1 -1123.3,E2 -1123.3} C_VEL
LIN {X 0,Y 594.353,Z 119.449,A -85,B 0,C 180,E1 -1126.162,E2 -1126.162} C_VEL
LIN {X 0,Y 594.37,Z 119.443,A -85,B 0,C 180,E1 -1129.179,E2 -1129.179} C_VEL
LIN {X 0,Y 594.375,Z 119.448,A -85,B 0,C 180,E1 -1132.06,E2 -1132.06} C_VEL
LIN {X 0,Y 594.347,Z 119.448,A -85,B 0,C 180,E1 -1134.677,E2 -1134.677} C_VEL
LIN {X 0,Y 594.372,Z 119.442,A -85,B 0,C 180,E1 -1137.09,E2 -1137.09} C_VEL
LIN {X 0,Y 594.385,Z 119.445,A -85,B 0,C 180,E1 -1139.673,E2 -1139.673} C_VEL
LIN {X 0,Y 594.373,Z 119.444,A -85,B 0,C 180,E1 -1142.54,E2 -1142.54} C_VEL
LIN {X 0,Y 594.372,Z 119.442,A -85,B 0,C 180,E1 -1144.808,E2 -1144.808} C_VEL
LIN {X 0,Y 594.402,Z 119.468,A -85,B 0,C 180,E1 -1146.575,E2 -1146.575} C_VEL
LIN {X 0,Y 594.813,Z 124.483,A -85,B 0,C 180,E1 -1147.283,E2 -1147.283} C_VEL
LIN {X 0,Y 594.677,Z 145.416,A -85,B 0,C 180,E1 -1150.138,E2 -1150.138} C_VEL
LIN {X 0,Y 594.566,Z 166.388,A -85,B 0,C 180,E1 -1152.95,E2 -1152.95} C_VEL
LIN {X 0,Y 594.447,Z 188.005,A -85,B 0,C 180,E1 -1155.806,E2 -1155.806} C_VEL
LIN {X 0,Y 594.426,Z 194.528,A -85,B 0,C 180,E1 -1156.66,E2 -1156.66} C_VEL
LIN {X 0,Y 594.732,Z 200.576,A -85,B 0,C 180,E1 -1156.743,E2 -1156.743} C_VEL
LIN {X 0,Y 594.664,Z 302.989,A -85,B 0,C 180,E1 -1158,E2 -1158} C_VEL
LIN {X 0,Y 594.601,Z 316.247,A -85,B 0,C 180,E1 -1158.301,E2 -1158.301} C_VEL
LIN {X 0,Y 594.563,Z 329.224,A -85,B 0,C 180,E1 -1158.743,E2 -1158.743} C_VEL
LIN {X 0,Y 594.536,Z 340.646,A -85,B 0,C 180,E1 -1159.271,E2 -1159.271} C_VEL
LIN {X 0,Y 594.477,Z 352.213,A -85,B 0,C 180,E1 -1159.958,E2 -1159.958} C_VEL
LIN {X 0,Y 594.414,Z 362.607,A -85,B 0,C 180,E1 -1160.73,E2 -1160.73} C_VEL
LIN {X 0,Y 594.383,Z 371.12,A -85,B 0,C 180,E1 -1161.501,E2 -1161.501} C_VEL
LIN {X 0,Y 594.347,Z 378.967,A -85,B 0,C 180,E1 -1162.356,E2 -1162.356} C_VEL
LIN {X 0,Y 594.282,Z 386.816,A -85,B 0,C 180,E1 -1163.409,E2 -1163.409} C_VEL
LIN {X 0,Y 594.289,Z 393.684,A -85,B 0,C 180,E1 -1164.572,E2 -1164.572} C_VEL
LIN {X 0,Y 594.27,Z 398.374,A -85,B 0,C 180,E1 -1165.592,E2 -1165.592} C_VEL
LIN {X 0,Y 594.267,Z 401.959,A -85,B 0,C 180,E1 -1166.611,E2 -1166.611} C_VEL
LIN {X 0,Y 594.226,Z 403.81,A -85,B 0,C 180,E1 -1167.289,E2 -1167.289} C_VEL
LIN {X 0,Y 594.242,Z 405.202,A -85,B 0,C 180,E1 -1167.967,E2 -1167.967} C_VEL
LIN {X 0,Y 594.239,Z 406.785,A -85,B 0,C 180,E1 -1169.323,E2 -1169.323} C_VEL
LIN {X 0,Y 594.236,Z 407,A -85,B 0,C 180,E1 -1170.001,E2 -1170.001} C_VEL
LIN {X 0,Y 594.247,Z 406.184,A -85,B 0,C 180,E1 -1171.356,E2 -1171.356} C_VEL
LIN {X 0,Y 594.242,Z 405.2,A -85,B 0,C 180,E1 -1172.034,E2 -1172.034} C_VEL
LIN {X 0,Y 594.226,Z 403.808,A -85,B 0,C 180,E1 -1172.712,E2 -1172.712} C_VEL
LIN {X 0,Y 594.289,Z 400.894,A -85,B 0,C 180,E1 -1173.73,E2 -1173.73} C_VEL
LIN {X 0,Y 594.241,Z 396.947,A -85,B 0,C 180,E1 -1174.749,E2 -1174.749} C_VEL
LIN {X 0,Y 594.305,Z 390.874,A -85,B 0,C 180,E1 -1175.94,E2 -1175.94} C_VEL
LIN {X 0,Y 594.308,Z 384.233,A -85,B 0,C 180,E1 -1176.963,E2 -1176.963} C_VEL
LIN {X 0,Y 594.359,Z 375.985,A -85,B 0,C 180,E1 -1177.987,E2 -1177.987} C_VEL
LIN {X 0,Y 594.382,Z 367.532,A -85,B 0,C 180,E1 -1178.843,E2 -1178.843} C_VEL
LIN {X 0,Y 594.432,Z 357.088,A -85,B 0,C 180,E1 -1179.7,E2 -1179.7} C_VEL
LIN {X 0,Y 594.482,Z 346.75,A -85,B 0,C 180,E1 -1180.387,E2 -1180.387} C_VEL
LIN {X 0,Y 594.558,Z 335.723,A -85,B 0,C 180,E1 -1180.973,E2 -1180.973} C_VEL
LIN {X 0,Y 594.579,Z 323.7,A -85,B 0,C 180,E1 -1181.465,E2 -1181.465} C_VEL
LIN {X 0,Y 594.624,Z 310.331,A -85,B 0,C 180,E1 -1181.851,E2 -1181.851} C_VEL
LIN {X 0,Y 594.694,Z 297.049,A -85,B 0,C 180,E1 -1182.087,E2 -1182.087} C_VEL
LIN {X 0,Y 594.621,Z 196.001,A -85,B 0,C 180,E1 -1183.315,E2 -1183.315} C_VEL
LIN {X 0,Y 594.415,Z 194.269,A -85,B 0,C 180,E1 -1183.374,E2 -1183.374} C_VEL
LIN {X 0,Y 594.536,Z 171.998,A -85,B 0,C 180,E1 -1186.305,E2 -1186.305} C_VEL
LIN {X 0,Y 594.58,Z 152.793,A -85,B 0,C 180,E1 -1188.87,E2 -1188.87} C_VEL
LIN {X 0,Y 594.769,Z 132.111,A -85,B 0,C 180,E1 -1191.67,E2 -1191.67} C_VEL
LIN {X 0,Y 594.755,Z 121.474,A -85,B 0,C 180,E1 -1193.136,E2 -1193.136} C_VEL
LIN {X 0,Y 594.377,Z 119.447,A -85,B 0,C 180,E1 -1193.451,E2 -1193.451} C_VEL
LIN {X 0,Y 594.365,Z 119.452,A -85,B 0,C 180,E1 -1196.018,E2 -1196.018} C_VEL
LIN {X 0,Y 594.367,Z 119.45,A -85,B 0,C 180,E1 -1198.228,E2 -1198.228} C_VEL
LIN {X 0,Y 594.37,Z 119.444,A -85,B 0,C 180,E1 -1200.56,E2 -1200.56} C_VEL
LIN {X 0,Y 594.378,Z 119.442,A -85,B 0,C 180,E1 -1202.95,E2 -1202.95} C_VEL
LIN {X 0,Y 594.349,Z 119.449,A -85,B 0,C 180,E1 -1205.409,E2 -1205.409} C_VEL
LIN {X 0,Y 594.377,Z 119.447,A -85,B 0,C 180,E1 -1207.942,E2 -1207.942} C_VEL
LIN {X 0,Y 594.375,Z 119.442,A -85,B 0,C 180,E1 -1210.821,E2 -1210.821} C_VEL
LIN {X 0,Y 594.361,Z 119.448,A -85,B 0,C 180,E1 -1213.839,E2 -1213.839} C_VEL
LIN {X 0,Y 594.351,Z 119.446,A -85,B 0,C 180,E1 -1216.699,E2 -1216.699} C_VEL
LIN {X 0,Y 594.359,Z 119.451,A -85,B 0,C 180,E1 -1219.432,E2 -1219.432} C_VEL
LIN {X 0,Y 594.383,Z 119.441,A -85,B 0,C 180,E1 -1222.392,E2 -1222.392} C_VEL
LIN {X 0,Y 594.371,Z 119.447,A -85,B 0,C 180,E1 -1225.419,E2 -1225.419} C_VEL
LIN {X 0,Y 594.366,Z 119.444,A -85,B 0,C 180,E1 -1228.359,E2 -1228.359} C_VEL
LIN {X 0,Y 594.37,Z 119.45,A -85,B 0,C 180,E1 -1231.044,E2 -1231.044} C_VEL
LIN {X 0,Y 594.371,Z 119.445,A -85,B 0,C 180,E1 -1233.3,E2 -1233.3} C_VEL
LIN {X 0,Y 594.342,Z 119.449,A -85,B 0,C 180,E1 -1236.294,E2 -1236.294} C_VEL
LIN {X 0,Y 594.37,Z 119.443,A -85,B 0,C 180,E1 -1239.223,E2 -1239.223} C_VEL
LIN {X 0,Y 594.318,Z 119.452,A -85,B 0,C 180,E1 -1242.094,E2 -1242.094} C_VEL
LIN {X 0,Y 594.328,Z 119.449,A -85,B 0,C 180,E1 -1244.921,E2 -1244.921} C_VEL
LIN {X 0,Y 594.338,Z 119.447,A -85,B 0,C 180,E1 -1247.711,E2 -1247.711} C_VEL
LIN {X 0,Y 594.334,Z 119.452,A -85,B 0,C 180,E1 -1250.471,E2 -1250.471} C_VEL
LIN {X 0,Y 594.336,Z 119.446,A -85,B 0,C 180,E1 -1253.209,E2 -1253.209} C_VEL
LIN {X 0,Y 594.341,Z 119.454,A -85,B 0,C 180,E1 -1255.932,E2 -1255.932} C_VEL
LIN {X 0,Y 594.333,Z 119.448,A -85,B 0,C 180,E1 -1258.645,E2 -1258.645} C_VEL
LIN {X 0,Y 594.317,Z 119.449,A -85,B 0,C 180,E1 -1260.678,E2 -1260.678} C_VEL
LIN {X 0,Y 594.362,Z 119.442,A -85,B 0,C 180,E1 -1262.711,E2 -1262.711} C_VEL
LIN {X 0,Y 594.366,Z 119.448,A -85,B 0,C 180,E1 -1265.428,E2 -1265.428} C_VEL
LIN {X 0,Y 594.37,Z 119.444,A -85,B 0,C 180,E1 -1268.157,E2 -1268.157} C_VEL
LIN {X 0,Y 594.363,Z 119.446,A -85,B 0,C 180,E1 -1271.061,E2 -1271.061} C_VEL
LIN {X 0,Y 594.362,Z 119.448,A -85,B 0,C 180,E1 -1273.68,E2 -1273.68} C_VEL
LIN {X 0,Y 594.332,Z 119.45,A -85,B 0,C 180,E1 -1275.283,E2 -1275.283} C_VEL
LIN {X 0,Y 593.661,Z 119.534,A -85,B 0,C 180,E1 -1275.849,E2 -1275.849} C_VEL
LIN {X 0,Y 590.796,Z 119.889,A -85,B 0,C 180,E1 -1276.767,E2 -1276.767} C_VEL
LIN {X 0,Y 588.385,Z 120.194,A -85,B 0,C 180,E1 -1277.505,E2 -1277.505} C_VEL
LIN {X 0,Y 587.361,Z 120.316,A -85,B 0,C 180,E1 -1278.075,E2 -1278.075} C_VEL
LIN {X 0,Y 587.283,Z 120.325,A -85,B 0,C 180,E1 -1278.268,E2 -1278.268} C_VEL
LIN {X 0,Y 587.331,Z 120.326,A -85,B 0,C 180,E1 -1281.038,E2 -1281.038} C_VEL
LIN {X 0,Y 587.29,Z 120.323,A -85,B 0,C 180,E1 -1284.009,E2 -1284.009} C_VEL
LIN {X 0,Y 587.307,Z 120.323,A -85,B 0,C 180,E1 -1286.28,E2 -1286.28} C_VEL
LIN {X 0,Y 587.345,Z 120.323,A -85,B 0,C 180,E1 -1289.133,E2 -1289.133} C_VEL
LIN {X 0,Y 587.34,Z 120.318,A -85,B 0,C 180,E1 -1291.835,E2 -1291.835} C_VEL
LIN {X 0,Y 587.343,Z 120.321,A -85,B 0,C 180,E1 -1294.347,E2 -1294.347} C_VEL
LIN {X 0,Y 587.342,Z 120.318,A -85,B 0,C 180,E1 -1297.608,E2 -1297.608} C_VEL
LIN {X 0,Y 587.31,Z 120.327,A -85,B 0,C 180,E1 -1300.255,E2 -1300.255} C_VEL
LIN {X 0,Y 587.308,Z 120.323,A -85,B 0,C 180,E1 -1303.117,E2 -1303.117} C_VEL
LIN {X 0,Y 587.315,Z 120.326,A -85,B 0,C 180,E1 -1306.049,E2 -1306.049} C_VEL
LIN {X 0,Y 587.337,Z 120.319,A -85,B 0,C 180,E1 -1308.925,E2 -1308.925} C_VEL
LIN {X 0,Y 587.327,Z 120.321,A -85,B 0,C 180,E1 -1311.52,E2 -1311.52} C_VEL
LIN {X 0,Y 587.293,Z 120.333,A -85,B 0,C 180,E1 -1314.1,E2 -1314.1} C_VEL
LIN {X 0,Y 587.336,Z 120.32,A -85,B 0,C 180,E1 -1316.603,E2 -1316.603} C_VEL
LIN {X 0,Y 587.34,Z 120.322,A -85,B 0,C 180,E1 -1319.49,E2 -1319.49} C_VEL
LIN {X 0,Y 587.346,Z 120.32,A -85,B 0,C 180,E1 -1322.309,E2 -1322.309} C_VEL
LIN {X 0,Y 587.335,Z 120.32,A -85,B 0,C 180,E1 -1324.483,E2 -1324.483} C_VEL
LIN {X 0,Y 587.389,Z 120.466,A -85,B 0,C 180,E1 -1326.799,E2 -1326.799} C_VEL
LIN {X 0,Y 587.381,Z 134.286,A -85,B 0,C 180,E1 -1329.331,E2 -1329.331} C_VEL
LIN {X 0,Y 587.308,Z 146.651,A -85,B 0,C 180,E1 -1331.568,E2 -1331.568} C_VEL
LIN {X 0,Y 587.845,Z 151.496,A -85,B 0,C 180,E1 -1331.642,E2 -1331.642} C_VEL
LIN {X 0,Y 587.697,Z 252.982,A -85,B 0,C 180,E1 -1332.9,E2 -1332.9} C_VEL
LIN {X 0,Y 587.612,Z 265.946,A -85,B 0,C 180,E1 -1333.197,E2 -1333.197} C_VEL
LIN {X 0,Y 587.595,Z 278.653,A -85,B 0,C 180,E1 -1333.631,E2 -1333.631} C_VEL
LIN {X 0,Y 587.516,Z 291.04,A -85,B 0,C 180,E1 -1334.208,E2 -1334.208} C_VEL
LIN {X 0,Y 587.446,Z 302.731,A -85,B 0,C 180,E1 -1334.917,E2 -1334.917} C_VEL
LIN {X 0,Y 587.386,Z 313.461,A -85,B 0,C 180,E1 -1335.734,E2 -1335.734} C_VEL
LIN {X 0,Y 587.334,Z 323.408,A -85,B 0,C 180,E1 -1336.682,E2 -1336.682} C_VEL
LIN {X 0,Y 587.259,Z 332.329,A -85,B 0,C 180,E1 -1337.735,E2 -1337.735} C_VEL
LIN {X 0,Y 587.263,Z 338.35,A -85,B 0,C 180,E1 -1338.611,E2 -1338.611} C_VEL
LIN {X 0,Y 587.183,Z 344.236,A -85,B 0,C 180,E1 -1339.657,E2 -1339.657} C_VEL
LIN {X 0,Y 587.19,Z 348.853,A -85,B 0,C 180,E1 -1340.701,E2 -1340.701} C_VEL
LIN {X 0,Y 587.177,Z 352.35,A -85,B 0,C 180,E1 -1341.742,E2 -1341.742} C_VEL
LIN {X 0,Y 587.152,Z 354.1,A -85,B 0,C 180,E1 -1342.434,E2 -1342.434} C_VEL
LIN {X 0,Y 587.189,Z 355.896,A -85,B 0,C 180,E1 -1343.425,E2 -1343.425} C_VEL
LIN {X 0,Y 587.17,Z 356.877,A -85,B 0,C 180,E1 -1344.505,E2 -1344.505} C_VEL
LIN {X 0,Y 587.171,Z 356.683,A -85,B 0,C 180,E1 -1345.881,E2 -1345.881} C_VEL
LIN {X 0,Y 587.181,Z 356.009,A -85,B 0,C 180,E1 -1346.568,E2 -1346.568} C_VEL
LIN {X 0,Y 587.129,Z 354.937,A -85,B 0,C 180,E1 -1347.255,E2 -1347.255} C_VEL
LIN {X 0,Y 587.142,Z 353.419,A -85,B 0,C 180,E1 -1347.941,E2 -1347.941} C_VEL
LIN {X 0,Y 587.165,Z 350.37,A -85,B 0,C 180,E1 -1348.971,E2 -1348.971} C_VEL
LIN {X 0,Y 587.189,Z 346.283,A -85,B 0,C 180,E1 -1349.999,E2 -1349.999} C_VEL
LIN {X 0,Y 587.262,Z 340.036,A -85,B 0,C 180,E1 -1351.199,E2 -1351.199} C_VEL
LIN {X 0,Y 587.256,Z 333.254,A -85,B 0,C 180,E1 -1352.228,E2 -1352.228} C_VEL
LIN {X 0,Y 587.275,Z 324.822,A -85,B 0,C 180,E1 -1353.258,E2 -1353.258} C_VEL
LIN {X 0,Y 587.329,Z 316.174,A -85,B 0,C 180,E1 -1354.116,E2 -1354.116} C_VEL
LIN {X 0,Y 587.401,Z 305.562,A -85,B 0,C 180,E1 -1354.976,E2 -1354.976} C_VEL
LIN {X 0,Y 587.501,Z 294.988,A -85,B 0,C 180,E1 -1355.663,E2 -1355.663} C_VEL
LIN {X 0,Y 587.612,Z 282.763,A -85,B 0,C 180,E1 -1356.284,E2 -1356.284} C_VEL
LIN {X 0,Y 587.609,Z 270.861,A -85,B 0,C 180,E1 -1356.743,E2 -1356.743} C_VEL
LIN {X 0,Y 587.691,Z 258.013,A -85,B 0,C 180,E1 -1357.093,E2 -1357.093} C_VEL
LIN {X 0,Y 587.715,Z 243.624,A -85,B 0,C 180,E1 -1357.32,E2 -1357.32} C_VEL
LIN {X 0,Y 587.841,Z 150.224,A -85,B 0,C 180,E1 -1358.464,E2 -1358.464} C_VEL
LIN {X 0,Y 587.326,Z 146.569,A -85,B 0,C 180,E1 -1358.537,E2 -1358.537} C_VEL
LIN {X 0,Y 587.422,Z 131.04,A -85,B 0,C 180,E1 -1361.35,E2 -1361.35} C_VEL
LIN {X 0,Y 587.345,Z 120.321,A -85,B 0,C 180,E1 -1363.338,E2 -1363.338} C_VEL
LIN {X 0,Y 587.321,Z 120.325,A -85,B 0,C 180,E1 -1365.974,E2 -1365.974} C_VEL
LIN {X 0,Y 587.344,Z 120.32,A -85,B 0,C 180,E1 -1368.848,E2 -1368.848} C_VEL
LIN {X 0,Y 587.321,Z 120.324,A -85,B 0,C 180,E1 -1371.773,E2 -1371.773} C_VEL
LIN {X 0,Y 587.351,Z 120.318,A -85,B 0,C 180,E1 -1374.757,E2 -1374.757} C_VEL
LIN {X 0,Y 587.325,Z 120.32,A -85,B 0,C 180,E1 -1377.045,E2 -1377.045} C_VEL
LIN {X 0,Y 587.341,Z 120.32,A -85,B 0,C 180,E1 -1379.379,E2 -1379.379} C_VEL
LIN {X 0,Y 587.342,Z 120.327,A -85,B 0,C 180,E1 -1381.835,E2 -1381.835} C_VEL
LIN {X 0,Y 587.34,Z 120.32,A -85,B 0,C 180,E1 -1384.346,E2 -1384.346} C_VEL
LIN {X 0,Y 587.339,Z 120.327,A -85,B 0,C 180,E1 -1387.607,E2 -1387.607} C_VEL
LIN {X 0,Y 587.31,Z 120.323,A -85,B 0,C 180,E1 -1390.253,E2 -1390.253} C_VEL
LIN {X 0,Y 587.307,Z 120.326,A -85,B 0,C 180,E1 -1393.117,E2 -1393.117} C_VEL
LIN {X 0,Y 587.303,Z 120.324,A -85,B 0,C 180,E1 -1396.047,E2 -1396.047} C_VEL
LIN {X 0,Y 587.326,Z 120.324,A -85,B 0,C 180,E1 -1398.924,E2 -1398.924} C_VEL
LIN {X 0,Y 587.311,Z 120.327,A -85,B 0,C 180,E1 -1401.519,E2 -1401.519} C_VEL
LIN {X 0,Y 587.279,Z 120.326,A -85,B 0,C 180,E1 -1404.099,E2 -1404.099} C_VEL
LIN {X 0,Y 587.325,Z 120.327,A -85,B 0,C 180,E1 -1406.888,E2 -1406.888} C_VEL
LIN {X 0,Y 587.31,Z 120.325,A -85,B 0,C 180,E1 -1409.492,E2 -1409.492} C_VEL
LIN {X 0,Y 587.339,Z 120.32,A -85,B 0,C 180,E1 -1412.307,E2 -1412.307} C_VEL
LIN {X 0,Y 587.291,Z 120.328,A -85,B 0,C 180,E1 -1415.239,E2 -1415.239} C_VEL
LIN {X 0,Y 587.301,Z 120.326,A -85,B 0,C 180,E1 -1418.225,E2 -1418.225} C_VEL
LIN {X 0,Y 587.314,Z 120.324,A -85,B 0,C 180,E1 -1421.15,E2 -1421.15} C_VEL
LIN {X 0,Y 587.283,Z 120.328,A -85,B 0,C 180,E1 -1424.023,E2 -1424.023} C_VEL
LIN {X 0,Y 587.325,Z 120.326,A -85,B 0,C 180,E1 -1426.153,E2 -1426.153} C_VEL
LIN {X 0,Y 587.324,Z 120.322,A -85,B 0,C 180,E1 -1428.962,E2 -1428.962} C_VEL
LIN {X 0,Y 587.32,Z 120.323,A -85,B 0,C 180,E1 -1431.744,E2 -1431.744} C_VEL
LIN {X 0,Y 587.328,Z 120.324,A -85,B 0,C 180,E1 -1434.507,E2 -1434.507} C_VEL
LIN {X 0,Y 587.321,Z 120.321,A -85,B 0,C 180,E1 -1437.256,E2 -1437.256} C_VEL
LIN {X 0,Y 587.369,Z 120.324,A -85,B 0,C 180,E1 -1440,E2 -1440} C_VEL
LIN {X 0,Y 587.323,Z 120.321,A -85,B 0,C 180,E1 -1442.743,E2 -1442.743} C_VEL
LIN {X 0,Y 587.33,Z 120.325,A -85,B 0,C 180,E1 -1445.493,E2 -1445.493} C_VEL
LIN {X 0,Y 587.322,Z 120.323,A -85,B 0,C 180,E1 -1448.256,E2 -1448.256} C_VEL
LIN {X 0,Y 587.317,Z 120.324,A -85,B 0,C 180,E1 -1451.125,E2 -1451.125} C_VEL
LIN {X 0,Y 587.326,Z 120.325,A -85,B 0,C 180,E1 -1453.847,E2 -1453.847} C_VEL
LIN {X 0,Y 587.312,Z 120.323,A -85,B 0,C 180,E1 -1456.807,E2 -1456.807} C_VEL
LIN {X 0,Y 587.293,Z 120.33,A -85,B 0,C 180,E1 -1459.577,E2 -1459.577} C_VEL
LIN {X 0,Y 587.301,Z 120.326,A -85,B 0,C 180,E1 -1461.775,E2 -1461.775} C_VEL
LIN {X 0,Y 587.292,Z 120.328,A -85,B 0,C 180,E1 -1464.761,E2 -1464.761} C_VEL
LIN {X 0,Y 587.339,Z 120.32,A -85,B 0,C 180,E1 -1467.693,E2 -1467.693} C_VEL
LIN {X 0,Y 587.315,Z 120.324,A -85,B 0,C 180,E1 -1470.509,E2 -1470.509} C_VEL
LIN {X 0,Y 587.325,Z 120.327,A -85,B 0,C 180,E1 -1473.112,E2 -1473.112} C_VEL
LIN {X 0,Y 587.288,Z 120.326,A -85,B 0,C 180,E1 -1475.539,E2 -1475.539} C_VEL
LIN {X 0,Y 587.324,Z 120.32,A -85,B 0,C 180,E1 -1477.839,E2 -1477.839} C_VEL
LIN {X 0,Y 587.301,Z 120.327,A -85,B 0,C 180,E1 -1480.256,E2 -1480.256} C_VEL
LIN {X 0,Y 587.308,Z 120.324,A -85,B 0,C 180,E1 -1483.119,E2 -1483.119} C_VEL
LIN {X 0,Y 587.305,Z 120.326,A -85,B 0,C 180,E1 -1486.049,E2 -1486.049} C_VEL
LIN {X 0,Y 587.33,Z 120.321,A -85,B 0,C 180,E1 -1488.926,E2 -1488.926} C_VEL
LIN {X 0,Y 587.319,Z 120.321,A -85,B 0,C 180,E1 -1491.521,E2 -1491.521} C_VEL
LIN {X 0,Y 587.286,Z 120.333,A -85,B 0,C 180,E1 -1494.101,E2 -1494.101} C_VEL
LIN {X 0,Y 587.331,Z 120.322,A -85,B 0,C 180,E1 -1496.604,E2 -1496.604} C_VEL
LIN {X 0,Y 587.338,Z 120.32,A -85,B 0,C 180,E1 -1499.49,E2 -1499.49} C_VEL
LIN {X 0,Y 587.349,Z 120.321,A -85,B 0,C 180,E1 -1502.308,E2 -1502.308} C_VEL
LIN {X 0,Y 587.332,Z 120.321,A -85,B 0,C 180,E1 -1504.484,E2 -1504.484} C_VEL
LIN {X 0,Y 587.381,Z 120.509,A -85,B 0,C 180,E1 -1506.465,E2 -1506.465} C_VEL
LIN {X 0,Y 587.865,Z 124.332,A -85,B 0,C 180,E1 -1507.006,E2 -1507.006} C_VEL
LIN {X 0,Y 587.749,Z 142.757,A -85,B 0,C 180,E1 -1509.529,E2 -1509.529} C_VEL
LIN {X 0,Y 587.606,Z 164.031,A -85,B 0,C 180,E1 -1512.423,E2 -1512.423} C_VEL
LIN {X 0,Y 587.457,Z 183.974,A -85,B 0,C 180,E1 -1515.096,E2 -1515.096} C_VEL
LIN {X 0,Y 587.401,Z 194.445,A -85,B 0,C 180,E1 -1516.487,E2 -1516.487} C_VEL
LIN {X 0,Y 587.84,Z 198.788,A -85,B 0,C 180,E1 -1516.563,E2 -1516.563} C_VEL
LIN {X 0,Y 587.724,Z 302.989,A -85,B 0,C 180,E1 -1517.856,E2 -1517.856} C_VEL
LIN {X 0,Y 587.654,Z 316.248,A -85,B 0,C 180,E1 -1518.161,E2 -1518.161} C_VEL
LIN {X 0,Y 587.623,Z 328.646,A -85,B 0,C 180,E1 -1518.586,E2 -1518.586} C_VEL
LIN {X 0,Y 587.557,Z 340.644,A -85,B 0,C 180,E1 -1519.142,E2 -1519.142} C_VEL
LIN {X 0,Y 587.464,Z 352.215,A -85,B 0,C 180,E1 -1519.837,E2 -1519.837} C_VEL
LIN {X 0,Y 587.394,Z 362.609,A -85,B 0,C 180,E1 -1520.619,E2 -1520.619} C_VEL
LIN {X 0,Y 587.321,Z 371.12,A -85,B 0,C 180,E1 -1521.398,E2 -1521.398} C_VEL
LIN {X 0,Y 587.273,Z 378.967,A -85,B 0,C 180,E1 -1522.263,E2 -1522.263} C_VEL
LIN {X 0,Y 587.232,Z 385.474,A -85,B 0,C 180,E1 -1523.127,E2 -1523.127} C_VEL
LIN {X 0,Y 587.237,Z 391.87,A -85,B 0,C 180,E1 -1524.162,E2 -1524.162} C_VEL
LIN {X 0,Y 587.147,Z 396.953,A -85,B 0,C 180,E1 -1525.194,E2 -1525.194} C_VEL
LIN {X 0,Y 587.213,Z 400.898,A -85,B 0,C 180,E1 -1526.226,E2 -1526.226} C_VEL
LIN {X 0,Y 587.132,Z 403.81,A -85,B 0,C 180,E1 -1527.256,E2 -1527.256} C_VEL
LIN {X 0,Y 587.141,Z 405.2,A -85,B 0,C 180,E1 -1527.943,E2 -1527.943} C_VEL
LIN {X 0,Y 587.14,Z 406.785,A -85,B 0,C 180,E1 -1529.315,E2 -1529.315} C_VEL
LIN {X 0,Y 587.137,Z 407,A -85,B 0,C 180,E1 -1530.001,E2 -1530.001} C_VEL
LIN {X 0,Y 587.147,Z 406.185,A -85,B 0,C 180,E1 -1531.372,E2 -1531.372} C_VEL
LIN {X 0,Y 587.141,Z 405.199,A -85,B 0,C 180,E1 -1532.059,E2 -1532.059} C_VEL
LIN {X 0,Y 587.132,Z 403.808,A -85,B 0,C 180,E1 -1532.745,E2 -1532.745} C_VEL
LIN {X 0,Y 587.213,Z 400.894,A -85,B 0,C 180,E1 -1533.775,E2 -1533.775} C_VEL
LIN {X 0,Y 587.147,Z 396.947,A -85,B 0,C 180,E1 -1534.807,E2 -1534.807} C_VEL
LIN {X 0,Y 587.218,Z 390.874,A -85,B 0,C 180,E1 -1536.012,E2 -1536.012} C_VEL
LIN {X 0,Y 587.245,Z 384.233,A -85,B 0,C 180,E1 -1537.047,E2 -1537.047} C_VEL
LIN {X 0,Y 587.3,Z 375.986,A -85,B 0,C 180,E1 -1538.084,E2 -1538.084} C_VEL
LIN {X 0,Y 587.344,Z 367.532,A -85,B 0,C 180,E1 -1538.949,E2 -1538.949} C_VEL
LIN {X 0,Y 587.419,Z 357.09,A -85,B 0,C 180,E1 -1539.817,E2 -1539.817} C_VEL
LIN {X 0,Y 587.497,Z 346.748,A -85,B 0,C 180,E1 -1540.512,E2 -1540.512} C_VEL
LIN {X 0,Y 587.561,Z 334.809,A -85,B 0,C 180,E1 -1541.149,E2 -1541.149} C_VEL
LIN {X 0,Y 587.63,Z 322.586,A -85,B 0,C 180,E1 -1541.64,E2 -1541.64} C_VEL
LIN {X 0,Y 587.705,Z 309.415,A -85,B 0,C 180,E1 -1542.014,E2 -1542.014} C_VEL
LIN {X 0,Y 587.777,Z 297.049,A -85,B 0,C 180,E1 -1542.232,E2 -1542.232} C_VEL
LIN {X 0,Y 587.714,Z 196.67,A -85,B 0,C 180,E1 -1543.466,E2 -1543.466} C_VEL
LIN {X 0,Y 587.402,Z 194.435,A -85,B 0,C 180,E1 -1543.514,E2 -1543.514} C_VEL
LIN {X 0,Y 587.557,Z 173.328,A -85,B 0,C 180,E1 -1546.326,E2 -1546.326} C_VEL
LIN {X 0,Y 587.62,Z 153.523,A -85,B 0,C 180,E1 -1549.002,E2 -1549.002} C_VEL
LIN {X 0,Y 587.851,Z 133.437,A -85,B 0,C 180,E1 -1551.754,E2 -1551.754} C_VEL
LIN {X 0,Y 587.732,Z 122.544,A -85,B 0,C 180,E1 -1553.242,E2 -1553.242} C_VEL
LIN {X 0,Y 587.343,Z 120.325,A -85,B 0,C 180,E1 -1553.585,E2 -1553.585} C_VEL
LIN {X 0,Y 587.312,Z 120.329,A -85,B 0,C 180,E1 -1556.28,E2 -1556.28} C_VEL
LIN {X 0,Y 587.347,Z 120.318,A -85,B 0,C 180,E1 -1559.132,E2 -1559.132} C_VEL
LIN {X 0,Y 587.341,Z 120.328,A -85,B 0,C 180,E1 -1561.835,E2 -1561.835} C_VEL
LIN {X 0,Y 587.343,Z 120.32,A -85,B 0,C 180,E1 -1564.347,E2 -1564.347} C_VEL
LIN {X 0,Y 587.343,Z 120.326,A -85,B 0,C 180,E1 -1567.608,E2 -1567.608} C_VEL
LIN {X 0,Y 587.312,Z 120.323,A -85,B 0,C 180,E1 -1570.255,E2 -1570.255} C_VEL
LIN {X 0,Y 587.303,Z 120.326,A -85,B 0,C 180,E1 -1573.117,E2 -1573.117} C_VEL
LIN {X 0,Y 587.299,Z 120.324,A -85,B 0,C 180,E1 -1576.047,E2 -1576.047} C_VEL
LIN {X 0,Y 587.332,Z 120.323,A -85,B 0,C 180,E1 -1578.926,E2 -1578.926} C_VEL
LIN {X 0,Y 587.315,Z 120.326,A -85,B 0,C 180,E1 -1581.519,E2 -1581.519} C_VEL
LIN {X 0,Y 587.285,Z 120.325,A -85,B 0,C 180,E1 -1584.099,E2 -1584.099} C_VEL
LIN {X 0,Y 587.332,Z 120.327,A -85,B 0,C 180,E1 -1586.889,E2 -1586.889} C_VEL
LIN {X 0,Y 587.306,Z 120.324,A -85,B 0,C 180,E1 -1589.495,E2 -1589.495} C_VEL
LIN {X 0,Y 587.288,Z 120.327,A -85,B 0,C 180,E1 -1591.401,E2 -1591.401} C_VEL
LIN {X 0,Y 587.303,Z 120.322,A -85,B 0,C 180,E1 -1593.83,E2 -1593.83} C_VEL
LIN {X 0,Y 587.291,Z 120.334,A -85,B 0,C 180,E1 -1596.74,E2 -1596.74} C_VEL
LIN {X 0,Y 587.312,Z 120.325,A -85,B 0,C 180,E1 -1598.967,E2 -1598.967} C_VEL
LIN {X 0,Y 587.318,Z 120.322,A -85,B 0,C 180,E1 -1601.15,E2 -1601.15} C_VEL
LIN {X 0,Y 587.28,Z 120.329,A -85,B 0,C 180,E1 -1604.024,E2 -1604.024} C_VEL
LIN {X 0,Y 587.329,Z 120.325,A -85,B 0,C 180,E1 -1606.154,E2 -1606.154} C_VEL
LIN {X 0,Y 587.288,Z 120.325,A -85,B 0,C 180,E1 -1608.961,E2 -1608.961} C_VEL
LIN {X 0,Y 587.308,Z 120.324,A -85,B 0,C 180,E1 -1611.744,E2 -1611.744} C_VEL
LIN {X 0,Y 587.323,Z 120.324,A -85,B 0,C 180,E1 -1614.507,E2 -1614.507} C_VEL
LIN {X 0,Y 587.329,Z 120.319,A -85,B 0,C 180,E1 -1617.257,E2 -1617.257} C_VEL
LIN {X 0,Y 587.377,Z 120.322,A -85,B 0,C 180,E1 -1620,E2 -1620} C_VEL
LIN {X 0,Y 587.331,Z 120.318,A -85,B 0,C 180,E1 -1622.744,E2 -1622.744} C_VEL
LIN {X 0,Y 587.334,Z 120.325,A -85,B 0,C 180,E1 -1625.493,E2 -1625.493} C_VEL
LIN {X 0,Y 587.329,Z 120.32,A -85,B 0,C 180,E1 -1628.256,E2 -1628.256} C_VEL
LIN {X 0,Y 587.329,Z 120.323,A -85,B 0,C 180,E1 -1631.124,E2 -1631.124} C_VEL
LIN {X 0,Y 587.317,Z 120.32,A -85,B 0,C 180,E1 -1634.242,E2 -1634.242} C_VEL
LIN {X 0,Y 587.322,Z 120.322,A -85,B 0,C 180,E1 -1636.806,E2 -1636.806} C_VEL
LIN {X 0,Y 587.283,Z 120.325,A -85,B 0,C 180,E1 -1638.268,E2 -1638.268} C_VEL
LIN {X 0,Y 586.646,Z 120.409,A -85,B 0,C 180,E1 -1638.84,E2 -1638.84} C_VEL
LIN {X 0,Y 583.845,Z 120.762,A -85,B 0,C 180,E1 -1639.769,E2 -1639.769} C_VEL
LIN {X 0,Y 581.446,Z 121.064,A -85,B 0,C 180,E1 -1640.516,E2 -1640.516} C_VEL
LIN {X 0,Y 580.386,Z 121.194,A -85,B 0,C 180,E1 -1641.093,E2 -1641.093} C_VEL
LIN {X 0,Y 580.285,Z 121.205,A -85,B 0,C 180,E1 -1641.288,E2 -1641.288} C_VEL
LIN {X 0,Y 580.252,Z 121.203,A -85,B 0,C 180,E1 -1643.559,E2 -1643.559} C_VEL
LIN {X 0,Y 580.266,Z 121.2,A -85,B 0,C 180,E1 -1646.329,E2 -1646.329} C_VEL
LIN {X 0,Y 580.287,Z 121.205,A -85,B 0,C 180,E1 -1648.977,E2 -1648.977} C_VEL
LIN {X 0,Y 580.3,Z 121.195,A -85,B 0,C 180,E1 -1652.03,E2 -1652.03} C_VEL
LIN {X 0,Y 580.289,Z 121.206,A -85,B 0,C 180,E1 -1654.697,E2 -1654.697} C_VEL
LIN {X 0,Y 580.298,Z 121.196,A -85,B 0,C 180,E1 -1657.269,E2 -1657.269} C_VEL
LIN {X 0,Y 580.289,Z 121.201,A -85,B 0,C 180,E1 -1660.27,E2 -1660.27} C_VEL
LIN {X 0,Y 580.276,Z 121.203,A -85,B 0,C 180,E1 -1662.707,E2 -1662.707} C_VEL
LIN {X 0,Y 580.261,Z 121.2,A -85,B 0,C 180,E1 -1665.611,E2 -1665.611} C_VEL
LIN {X 0,Y 580.276,Z 121.208,A -85,B 0,C 180,E1 -1668.231,E2 -1668.231} C_VEL
LIN {X 0,Y 580.287,Z 121.197,A -85,B 0,C 180,E1 -1670.966,E2 -1670.966} C_VEL
LIN {X 0,Y 580.27,Z 121.202,A -85,B 0,C 180,E1 -1673.596,E2 -1673.596} C_VEL
LIN {X 0,Y 580.317,Z 121.2,A -85,B 0,C 180,E1 -1676.145,E2 -1676.145} C_VEL
LIN {X 0,Y 580.278,Z 121.199,A -85,B 0,C 180,E1 -1678.614,E2 -1678.614} C_VEL
LIN {X 0,Y 580.292,Z 121.197,A -85,B 0,C 180,E1 -1681.024,E2 -1681.024} C_VEL
LIN {X 0,Y 580.295,Z 121.206,A -85,B 0,C 180,E1 -1683.666,E2 -1683.666} C_VEL
LIN {X 0,Y 580.297,Z 121.199,A -85,B 0,C 180,E1 -1686.442,E2 -1686.442} C_VEL
LIN {X 0,Y 580.354,Z 121.402,A -85,B 0,C 180,E1 -1686.745,E2 -1686.745} C_VEL
LIN {X 0,Y 580.361,Z 134.238,A -85,B 0,C 180,E1 -1689.127,E2 -1689.127} C_VEL
LIN {X 0,Y 580.28,Z 146.608,A -85,B 0,C 180,E1 -1691.394,E2 -1691.394} C_VEL
LIN {X 0,Y 580.963,Z 151.894,A -85,B 0,C 180,E1 -1691.485,E2 -1691.485} C_VEL
LIN {X 0,Y 580.756,Z 252.687,A -85,B 0,C 180,E1 -1692.747,E2 -1692.747} C_VEL
LIN {X 0,Y 580.653,Z 265.629,A -85,B 0,C 180,E1 -1693.043,E2 -1693.043} C_VEL
LIN {X 0,Y 580.635,Z 278.199,A -85,B 0,C 180,E1 -1693.474,E2 -1693.474} C_VEL
LIN {X 0,Y 580.562,Z 289.89,A -85,B 0,C 180,E1 -1694.014,E2 -1694.014} C_VEL
LIN {X 0,Y 580.443,Z 301.813,A -85,B 0,C 180,E1 -1694.731,E2 -1694.731} C_VEL
LIN {X 0,Y 580.35,Z 312.566,A -85,B 0,C 180,E1 -1695.545,E2 -1695.545} C_VEL
LIN {X 0,Y 580.314,Z 321.131,A -85,B 0,C 180,E1 -1696.34,E2 -1696.34} C_VEL
LIN {X 0,Y 580.228,Z 329.087,A -85,B 0,C 180,E1 -1697.229,E2 -1697.229} C_VEL
LIN {X 0,Y 580.172,Z 336.817,A -85,B 0,C 180,E1 -1698.293,E2 -1698.293} C_VEL
LIN {X 0,Y 580.113,Z 343.919,A -85,B 0,C 180,E1 -1699.529,E2 -1699.529} C_VEL
LIN {X 0,Y 580.085,Z 348.607,A -85,B 0,C 180,E1 -1700.586,E2 -1700.586} C_VEL
LIN {X 0,Y 580.093,Z 352.165,A -85,B 0,C 180,E1 -1701.64,E2 -1701.64} C_VEL
LIN {X 0,Y 580.076,Z 353.972,A -85,B 0,C 180,E1 -1702.341,E2 -1702.341} C_VEL
LIN {X 0,Y 580.068,Z 356.279,A -85,B 0,C 180,E1 -1703.739,E2 -1703.739} C_VEL
LIN {X 0,Y 580.09,Z 356.843,A -85,B 0,C 180,E1 -1704.437,E2 -1704.437} C_VEL
LIN {X 0,Y 580.029,Z 356.986,A -85,B 0,C 180,E1 -1705.134,E2 -1705.134} C_VEL
LIN {X 0,Y 580.088,Z 356.724,A -85,B 0,C 180,E1 -1705.831,E2 -1705.831} C_VEL
LIN {X 0,Y 580.107,Z 356.078,A -85,B 0,C 180,E1 -1706.527,E2 -1706.527} C_VEL
LIN {X 0,Y 580.04,Z 355.046,A -85,B 0,C 180,E1 -1707.221,E2 -1707.221} C_VEL
LIN {X 0,Y 580.041,Z 353.574,A -85,B 0,C 180,E1 -1707.916,E2 -1707.916} C_VEL
LIN {X 0,Y 580.085,Z 350.585,A -85,B 0,C 180,E1 -1708.958,E2 -1708.958} C_VEL
LIN {X 0,Y 580.095,Z 346.564,A -85,B 0,C 180,E1 -1709.999,E2 -1709.999} C_VEL
LIN {X 0,Y 580.198,Z 340.387,A -85,B 0,C 180,E1 -1711.214,E2 -1711.214} C_VEL
LIN {X 0,Y 580.197,Z 333.684,A -85,B 0,C 180,E1 -1712.256,E2 -1712.256} C_VEL
LIN {X 0,Y 580.217,Z 325.382,A -85,B 0,C 180,E1 -1713.298,E2 -1713.298} C_VEL
LIN {X 0,Y 580.289,Z 316.848,A -85,B 0,C 180,E1 -1714.167,E2 -1714.167} C_VEL
LIN {X 0,Y 580.382,Z 306.373,A -85,B 0,C 180,E1 -1715.036,E2 -1715.036} C_VEL
LIN {X 0,Y 580.505,Z 295.99,A -85,B 0,C 180,E1 -1715.732,E2 -1715.732} C_VEL
LIN {X 0,Y 580.649,Z 284.021,A -85,B 0,C 180,E1 -1716.364,E2 -1716.364} C_VEL
LIN {X 0,Y 580.654,Z 272.65,A -85,B 0,C 180,E1 -1716.825,E2 -1716.825} C_VEL
LIN {X 0,Y 580.745,Z 259.666,A -85,B 0,C 180,E1 -1717.2,E2 -1717.2} C_VEL
LIN {X 0,Y 580.783,Z 246.603,A -85,B 0,C 180,E1 -1717.432,E2 -1717.432} C_VEL
LIN {X 0,Y 580.831,Z 149.932,A -85,B 0,C 180,E1 -1718.633,E2 -1718.633} C_VEL
LIN {X 0,Y 580.259,Z 146.552,A -85,B 0,C 180,E1 -1718.707,E2 -1718.707} C_VEL
LIN {X 0,Y 580.383,Z 131.386,A -85,B 0,C 180,E1 -1721.489,E2 -1721.489} C_VEL
LIN {X 0,Y 580.281,Z 121.201,A -85,B 0,C 180,E1 -1723.392,E2 -1723.392} C_VEL
LIN {X 0,Y 580.272,Z 121.206,A -85,B 0,C 180,E1 -1726.174,E2 -1726.174} C_VEL
LIN {X 0,Y 580.298,Z 121.195,A -85,B 0,C 180,E1 -1729.15,E2 -1729.15} C_VEL
LIN {X 0,Y 580.272,Z 121.206,A -85,B 0,C 180,E1 -1732.052,E2 -1732.052} C_VEL
LIN {X 0,Y 580.306,Z 121.194,A -85,B 0,C 180,E1 -1735.079,E2 -1735.079} C_VEL
LIN {X 0,Y 580.29,Z 121.203,A -85,B 0,C 180,E1 -1738.185,E2 -1738.185} C_VEL
LIN {X 0,Y 580.282,Z 121.198,A -85,B 0,C 180,E1 -1740.693,E2 -1740.693} C_VEL
LIN {X 0,Y 580.3,Z 121.198,A -85,B 0,C 180,E1 -1743.315,E2 -1743.315} C_VEL
LIN {X 0,Y 580.242,Z 121.212,A -85,B 0,C 180,E1 -1745.755,E2 -1745.755} C_VEL
LIN {X 0,Y 580.281,Z 121.201,A -85,B 0,C 180,E1 -1748.145,E2 -1748.145} C_VEL
LIN {X 0,Y 580.293,Z 121.197,A -85,B 0,C 180,E1 -1750.842,E2 -1750.842} C_VEL
LIN {X 0,Y 580.266,Z 121.207,A -85,B 0,C 180,E1 -1753.657,E2 -1753.657} C_VEL
LIN {X 0,Y 580.261,Z 121.201,A -85,B 0,C 180,E1 -1756.609,E2 -1756.609} C_VEL
LIN {X 0,Y 580.288,Z 121.204,A -85,B 0,C 180,E1 -1759.155,E2 -1759.155} C_VEL
LIN {X 0,Y 580.277,Z 121.199,A -85,B 0,C 180,E1 -1761.927,E2 -1761.927} C_VEL
LIN {X 0,Y 580.241,Z 121.204,A -85,B 0,C 180,E1 -1764.452,E2 -1764.452} C_VEL
LIN {X 0,Y 580.276,Z 121.207,A -85,B 0,C 180,E1 -1766.974,E2 -1766.974} C_VEL
LIN {X 0,Y 580.272,Z 121.202,A -85,B 0,C 180,E1 -1769.423,E2 -1769.423} C_VEL
LIN {X 0,Y 580.283,Z 121.198,A -85,B 0,C 180,E1 -1772.141,E2 -1772.141} C_VEL
LIN {X 0,Y 580.271,Z 121.207,A -85,B 0,C 180,E1 -1774.918,E2 -1774.918} C_VEL
LIN {X 0,Y 580.243,Z 121.203,A -85,B 0,C 180,E1 -1777.946,E2 -1777.946} C_VEL
LIN {X 0,Y 580.284,Z 121.203,A -85,B 0,C 180,E1 -1780.849,E2 -1780.849} C_VEL
LIN {X 0,Y 580.23,Z 121.205,A -85,B 0,C 180,E1 -1783.824,E2 -1783.824} C_VEL
LIN {X 0,Y 580.282,Z 121.201,A -85,B 0,C 180,E1 -1785.982,E2 -1785.982} C_VEL
LIN {X 0,Y 580.292,Z 121.199,A -85,B 0,C 180,E1 -1788.827,E2 -1788.827} C_VEL
LIN {X 0,Y 580.288,Z 121.199,A -85,B 0,C 180,E1 -1791.643,E2 -1791.643} C_VEL
LIN {X 0,Y 580.297,Z 121.201,A -85,B 0,C 180,E1 -1794.44,E2 -1794.44} C_VEL
LIN {X 0,Y 580.332,Z 121.199,A -85,B 0,C 180,E1 -1797.918,E2 -1797.918} C_VEL
LIN {X 0,Y 580.337,Z 121.2,A -85,B 0,C 180,E1 -1800,E2 -1800} C_VEL
LIN {X 0,Y 580.291,Z 121.197,A -85,B 0,C 180,E1 -1802.777,E2 -1802.777} C_VEL
LIN {X 0,Y 580.299,Z 121.202,A -85,B 0,C 180,E1 -1805.56,E2 -1805.56} C_VEL
LIN {X 0,Y 580.289,Z 121.198,A -85,B 0,C 180,E1 -1808.357,E2 -1808.357} C_VEL
LIN {X 0,Y 580.287,Z 121.2,A -85,B 0,C 180,E1 -1811.191,E2 -1811.191} C_VEL
LIN {X 0,Y 580.282,Z 121.2,A -85,B 0,C 180,E1 -1814.018,E2 -1814.018} C_VEL
LIN {X 0,Y 580.277,Z 121.201,A -85,B 0,C 180,E1 -1816.907,E2 -1816.907} C_VEL
LIN {X 0,Y 580.266,Z 121.202,A -85,B 0,C 180,E1 -1819.824,E2 -1819.824} C_VEL
LIN {X 0,Y 580.243,Z 121.203,A -85,B 0,C 180,E1 -1822.054,E2 -1822.054} C_VEL
LIN {X 0,Y 580.271,Z 121.208,A -85,B 0,C 180,E1 -1825.081,E2 -1825.081} C_VEL
LIN {X 0,Y 580.283,Z 121.198,A -85,B 0,C 180,E1 -1827.859,E2 -1827.859} C_VEL
LIN {X 0,Y 580.269,Z 121.204,A -85,B 0,C 180,E1 -1830.694,E2 -1830.694} C_VEL
LIN {X 0,Y 580.272,Z 121.202,A -85,B 0,C 180,E1 -1833.314,E2 -1833.314} C_VEL
LIN {X 0,Y 580.235,Z 121.203,A -85,B 0,C 180,E1 -1835.757,E2 -1835.757} C_VEL
LIN {X 0,Y 580.276,Z 121.2,A -85,B 0,C 180,E1 -1838.147,E2 -1838.147} C_VEL
LIN {X 0,Y 580.288,Z 121.203,A -85,B 0,C 180,E1 -1840.844,E2 -1840.844} C_VEL
LIN {X 0,Y 580.271,Z 121.199,A -85,B 0,C 180,E1 -1843.659,E2 -1843.659} C_VEL
LIN {X 0,Y 580.267,Z 121.207,A -85,B 0,C 180,E1 -1846.611,E2 -1846.611} C_VEL
LIN {X 0,Y 580.293,Z 121.196,A -85,B 0,C 180,E1 -1849.158,E2 -1849.158} C_VEL
LIN {X 0,Y 580.282,Z 121.202,A -85,B 0,C 180,E1 -1851.928,E2 -1851.928} C_VEL
LIN {X 0,Y 580.247,Z 121.207,A -85,B 0,C 180,E1 -1854.454,E2 -1854.454} C_VEL
LIN {X 0,Y 580.286,Z 121.197,A -85,B 0,C 180,E1 -1856.976,E2 -1856.976} C_VEL
LIN {X 0,Y 580.298,Z 121.197,A -85,B 0,C 180,E1 -1859.426,E2 -1859.426} C_VEL
LIN {X 0,Y 580.295,Z 121.203,A -85,B 0,C 180,E1 -1862.142,E2 -1862.142} C_VEL
LIN {X 0,Y 580.32,Z 121.194,A -85,B 0,C 180,E1 -1865.271,E2 -1865.271} C_VEL
LIN {X 0,Y 580.322,Z 121.217,A -85,B 0,C 180,E1 -1866.303,E2 -1866.303} C_VEL
LIN {X 0,Y 580.946,Z 125.79,A -85,B 0,C 180,E1 -1866.962,E2 -1866.962} C_VEL
LIN {X 0,Y 580.815,Z 145.358,A -85,B 0,C 180,E1 -1869.643,E2 -1869.643} C_VEL
LIN {X 0,Y 580.623,Z 165.36,A -85,B 0,C 180,E1 -1872.387,E2 -1872.387} C_VEL
LIN {X 0,Y 580.455,Z 185.304,A -85,B 0,C 180,E1 -1875.092,E2 -1875.092} C_VEL
LIN {X 0,Y 580.407,Z 194.528,A -85,B 0,C 180,E1 -1876.332,E2 -1876.332} C_VEL
LIN {X 0,Y 580.957,Z 200.576,A -85,B 0,C 180,E1 -1876.423,E2 -1876.423} C_VEL
LIN {X 0,Y 580.784,Z 302.989,A -85,B 0,C 180,E1 -1877.708,E2 -1877.708} C_VEL
LIN {X 0,Y 580.726,Z 316.247,A -85,B 0,C 180,E1 -1878.018,E2 -1878.018} C_VEL
LIN {X 0,Y 580.653,Z 329.164,A -85,B 0,C 180,E1 -1878.467,E2 -1878.467} C_VEL
LIN {X 0,Y 580.579,Z 340.642,A -85,B 0,C 180,E1 -1879.01,E2 -1879.01} C_VEL
LIN {X 0,Y 580.44,Z 352.212,A -85,B 0,C 180,E1 -1879.713,E2 -1879.713} C_VEL
LIN {X 0,Y 580.345,Z 362.61,A -85,B 0,C 180,E1 -1880.504,E2 -1880.504} C_VEL
LIN {X 0,Y 580.271,Z 371.12,A -85,B 0,C 180,E1 -1881.293,E2 -1881.293} C_VEL
LIN {X 0,Y 580.221,Z 378.967,A -85,B 0,C 180,E1 -1882.169,E2 -1882.169} C_VEL
LIN {X 0,Y 580.153,Z 386.654,A -85,B 0,C 180,E1 -1883.222,E2 -1883.222} C_VEL
LIN {X 0,Y 580.139,Z 393.684,A -85,B 0,C 180,E1 -1884.439,E2 -1884.439} C_VEL
LIN {X 0,Y 580.108,Z 398.375,A -85,B 0,C 180,E1 -1885.484,E2 -1885.484} C_VEL
LIN {X 0,Y 580.123,Z 401.959,A -85,B 0,C 180,E1 -1886.528,E2 -1886.528} C_VEL
LIN {X 0,Y 580.043,Z 403.81,A -85,B 0,C 180,E1 -1887.223,E2 -1887.223} C_VEL
LIN {X 0,Y 580.04,Z 405.199,A -85,B 0,C 180,E1 -1887.918,E2 -1887.918} C_VEL
LIN {X 0,Y 580.04,Z 406.785,A -85,B 0,C 180,E1 -1889.306,E2 -1889.306} C_VEL
LIN {X 0,Y 580.037,Z 407,A -85,B 0,C 180,E1 -1890.001,E2 -1890.001} C_VEL
LIN {X 0,Y 580.047,Z 406.186,A -85,B 0,C 180,E1 -1891.389,E2 -1891.389} C_VEL
LIN {X 0,Y 580.04,Z 405.198,A -85,B 0,C 180,E1 -1892.084,E2 -1892.084} C_VEL
LIN {X 0,Y 580.043,Z 403.808,A -85,B 0,C 180,E1 -1892.779,E2 -1892.779} C_VEL
LIN {X 0,Y 580.11,Z 400.894,A -85,B 0,C 180,E1 -1893.821,E2 -1893.821} C_VEL
LIN {X 0,Y 580.053,Z 396.947,A -85,B 0,C 180,E1 -1894.866,E2 -1894.866} C_VEL
LIN {X 0,Y 580.139,Z 390.874,A -85,B 0,C 180,E1 -1896.085,E2 -1896.085} C_VEL
LIN {X 0,Y 580.185,Z 384.234,A -85,B 0,C 180,E1 -1897.133,E2 -1897.133} C_VEL
LIN {X 0,Y 580.251,Z 375.986,A -85,B 0,C 180,E1 -1898.182,E2 -1898.182} C_VEL
LIN {X 0,Y 580.308,Z 367.533,A -85,B 0,C 180,E1 -1899.059,E2 -1899.059} C_VEL
LIN {X 0,Y 580.422,Z 357.091,A -85,B 0,C 180,E1 -1899.936,E2 -1899.936} C_VEL
LIN {X 0,Y 580.506,Z 346.746,A -85,B 0,C 180,E1 -1900.64,E2 -1900.64} C_VEL
LIN {X 0,Y 580.597,Z 335.239,A -85,B 0,C 180,E1 -1901.264,E2 -1901.264} C_VEL
LIN {X 0,Y 580.683,Z 322.457,A -85,B 0,C 180,E1 -1901.785,E2 -1901.785} C_VEL
LIN {X 0,Y 580.753,Z 309.413,A -85,B 0,C 180,E1 -1902.16,E2 -1902.16} C_VEL
LIN {X 0,Y 580.839,Z 297.049,A -85,B 0,C 180,E1 -1902.38,E2 -1902.38} C_VEL
LIN {X 0,Y 580.802,Z 197.343,A -85,B 0,C 180,E1 -1903.621,E2 -1903.621} C_VEL
LIN {X 0,Y 580.413,Z 194.435,A -85,B 0,C 180,E1 -1903.68,E2 -1903.68} C_VEL
LIN {X 0,Y 580.572,Z 171.998,A -85,B 0,C 180,E1 -1906.709,E2 -1906.709} C_VEL
LIN {X 0,Y 580.74,Z 151.812,A -85,B 0,C 180,E1 -1909.473,E2 -1909.473} C_VEL
LIN {X 0,Y 580.922,Z 130.389,A -85,B 0,C 180,E1 -1912.401,E2 -1912.401} C_VEL
LIN {X 0,Y 580.798,Z 124.006,A -85,B 0,C 180,E1 -1913.288,E2 -1913.288} C_VEL
LIN {X 0,Y 580.307,Z 121.202,A -85,B 0,C 180,E1 -1913.699,E2 -1913.699} C_VEL
LIN {X 0,Y 580.27,Z 121.206,A -85,B 0,C 180,E1 -1916.329,E2 -1916.329} C_VEL
LIN {X 0,Y 580.289,Z 121.198,A -85,B 0,C 180,E1 -1918.977,E2 -1918.977} C_VEL
LIN {X 0,Y 580.301,Z 121.203,A -85,B 0,C 180,E1 -1922.03,E2 -1922.03} C_VEL
LIN {X 0,Y 580.288,Z 121.197,A -85,B 0,C 180,E1 -1924.697,E2 -1924.697} C_VEL
LIN {X 0,Y 580.29,Z 121.199,A -85,B 0,C 180,E1 -1927.269,E2 -1927.269} C_VEL
LIN {X 0,Y 580.292,Z 121.197,A -85,B 0,C 180,E1 -1930.27,E2 -1930.27} C_VEL
LIN {X 0,Y 580.261,Z 121.2,A -85,B 0,C 180,E1 -1932.708,E2 -1932.708} C_VEL
LIN {X 0,Y 580.251,Z 121.208,A -85,B 0,C 180,E1 -1935.611,E2 -1935.611} C_VEL
LIN {X 0,Y 580.257,Z 121.201,A -85,B 0,C 180,E1 -1938.229,E2 -1938.229} C_VEL
LIN {X 0,Y 580.268,Z 121.204,A -85,B 0,C 180,E1 -1940.964,E2 -1940.964} C_VEL
LIN {X 0,Y 580.248,Z 121.205,A -85,B 0,C 180,E1 -1943.595,E2 -1943.595} C_VEL
LIN {X 0,Y 580.273,Z 121.199,A -85,B 0,C 180,E1 -1946.142,E2 -1946.142} C_VEL
LIN {X 0,Y 580.264,Z 121.204,A -85,B 0,C 180,E1 -1948.614,E2 -1948.614} C_VEL
LIN {X 0,Y 580.275,Z 121.206,A -85,B 0,C 180,E1 -1951.023,E2 -1951.023} C_VEL
LIN {X 0,Y 580.262,Z 121.2,A -85,B 0,C 180,E1 -1953.672,E2 -1953.672} C_VEL
LIN {X 0,Y 580.243,Z 121.207,A -85,B 0,C 180,E1 -1956.44,E2 -1956.44} C_VEL
LIN {X 0,Y 580.248,Z 121.201,A -85,B 0,C 180,E1 -1959.436,E2 -1959.436} C_VEL
LIN {X 0,Y 580.23,Z 121.203,A -85,B 0,C 180,E1 -1961.644,E2 -1961.644} C_VEL
LIN {X 0,Y 580.26,Z 121.207,A -85,B 0,C 180,E1 -1964.546,E2 -1964.546} C_VEL
LIN {X 0,Y 580.226,Z 121.208,A -85,B 0,C 180,E1 -1966.695,E2 -1966.695} C_VEL
LIN {X 0,Y 580.266,Z 121.201,A -85,B 0,C 180,E1 -1968.826,E2 -1968.826} C_VEL
LIN {X 0,Y 580.278,Z 121.199,A -85,B 0,C 180,E1 -1971.643,E2 -1971.643} C_VEL
LIN {X 0,Y 580.292,Z 121.2,A -85,B 0,C 180,E1 -1974.44,E2 -1974.44} C_VEL
LIN {X 0,Y 580.337,Z 121.198,A -85,B 0,C 180,E1 -1977.918,E2 -1977.918} C_VEL
LIN {X 0,Y 580.346,Z 121.197,A -85,B 0,C 180,E1 -1980,E2 -1980} C_VEL
LIN {X 0,Y 580.3,Z 121.194,A -85,B 0,C 180,E1 -1982.777,E2 -1982.777} C_VEL
LIN {X 0,Y 580.302,Z 121.202,A -85,B 0,C 180,E1 -1985.56,E2 -1985.56} C_VEL
LIN {X 0,Y 580.298,Z 121.195,A -85,B 0,C 180,E1 -1988.357,E2 -1988.357} C_VEL
LIN {X 0,Y 580.3,Z 121.199,A -85,B 0,C 180,E1 -1991.191,E2 -1991.191} C_VEL
LIN {X 0,Y 580.293,Z 121.196,A -85,B 0,C 180,E1 -1994.018,E2 -1994.018} C_VEL
LIN {X 0,Y 580.29,Z 121.2,A -85,B 0,C 180,E1 -1996.906,E2 -1996.906} C_VEL
LIN {X 0,Y 580.276,Z 121.199,A -85,B 0,C 180,E1 -1999.824,E2 -1999.824} C_VEL
LIN {X 0,Y 580.285,Z 121.205,A -85,B 0,C 180,E1 -2001.288,E2 -2001.288} C_VEL
LIN {X 0,Y 579.571,Z 121.29,A -85,B 0,C 180,E1 -2001.867,E2 -2001.867} C_VEL
LIN {X 0,Y 576.685,Z 121.65,A -85,B 0,C 180,E1 -2002.807,E2 -2002.807} C_VEL
LIN {X 0,Y 574.284,Z 121.946,A -85,B 0,C 180,E1 -2003.563,E2 -2003.563} C_VEL
LIN {X 0,Y 573.272,Z 122.07,A -85,B 0,C 180,E1 -2004.147,E2 -2004.147} C_VEL
LIN {X 0,Y 573.198,Z 122.079,A -85,B 0,C 180,E1 -2004.344,E2 -2004.344} C_VEL
LIN {X 0,Y 573.212,Z 122.088,A -85,B 0,C 180,E1 -2006.978,E2 -2006.978} C_VEL
LIN {X 0,Y 573.225,Z 122.078,A -85,B 0,C 180,E1 -2009.484,E2 -2009.484} C_VEL
LIN {X 0,Y 573.248,Z 122.075,A -85,B 0,C 180,E1 -2012.228,E2 -2012.228} C_VEL
LIN {X 0,Y 573.235,Z 122.084,A -85,B 0,C 180,E1 -2014.771,E2 -2014.771} C_VEL
LIN {X 0,Y 573.233,Z 122.076,A -85,B 0,C 180,E1 -2017.808,E2 -2017.808} C_VEL
LIN {X 0,Y 573.247,Z 122.08,A -85,B 0,C 180,E1 -2020.525,E2 -2020.525} C_VEL
LIN {X 0,Y 573.234,Z 122.075,A -85,B 0,C 180,E1 -2023.36,E2 -2023.36} C_VEL
LIN {X 0,Y 573.239,Z 122.084,A -85,B 0,C 180,E1 -2026.332,E2 -2026.332} C_VEL
LIN {X 0,Y 573.229,Z 122.081,A -85,B 0,C 180,E1 -2028.543,E2 -2028.543} C_VEL
LIN {X 0,Y 573.248,Z 122.074,A -85,B 0,C 180,E1 -2031.299,E2 -2031.299} C_VEL
LIN {X 0,Y 573.216,Z 122.087,A -85,B 0,C 180,E1 -2034.019,E2 -2034.019} C_VEL
LIN {X 0,Y 573.274,Z 122.072,A -85,B 0,C 180,E1 -2036.518,E2 -2036.518} C_VEL
LIN {X 0,Y 573.232,Z 122.076,A -85,B 0,C 180,E1 -2039.118,E2 -2039.118} C_VEL
LIN {X 0,Y 573.237,Z 122.08,A -85,B 0,C 180,E1 -2041.435,E2 -2041.435} C_VEL
LIN {X 0,Y 573.257,Z 122.074,A -85,B 0,C 180,E1 -2044.59,E2 -2044.59} C_VEL
LIN {X 0,Y 573.278,Z 122.136,A -85,B 0,C 180,E1 -2046.663,E2 -2046.663} C_VEL
LIN {X 0,Y 573.406,Z 131.556,A -85,B 0,C 180,E1 -2048.426,E2 -2048.426} C_VEL
LIN {X 0,Y 573.24,Z 146.714,A -85,B 0,C 180,E1 -2051.233,E2 -2051.233} C_VEL
LIN {X 0,Y 574.081,Z 153.347,A -85,B 0,C 180,E1 -2051.337,E2 -2051.337} C_VEL
LIN {X 0,Y 573.829,Z 253.706,A -85,B 0,C 180,E1 -2052.616,E2 -2052.616} C_VEL
LIN {X 0,Y 573.732,Z 267.445,A -85,B 0,C 180,E1 -2052.95,E2 -2052.95} C_VEL
LIN {X 0,Y 573.682,Z 280.001,A -85,B 0,C 180,E1 -2053.405,E2 -2053.405} C_VEL
LIN {X 0,Y 573.551,Z 292.007,A -85,B 0,C 180,E1 -2053.996,E2 -2053.996} C_VEL
LIN {X 0,Y 573.438,Z 303.517,A -85,B 0,C 180,E1 -2054.722,E2 -2054.722} C_VEL
LIN {X 0,Y 573.311,Z 314.164,A -85,B 0,C 180,E1 -2055.566,E2 -2055.566} C_VEL
LIN {X 0,Y 573.257,Z 323.904,A -85,B 0,C 180,E1 -2056.53,E2 -2056.53} C_VEL
LIN {X 0,Y 573.114,Z 332.724,A -85,B 0,C 180,E1 -2057.607,E2 -2057.607} C_VEL
LIN {X 0,Y 573.077,Z 339.728,A -85,B 0,C 180,E1 -2058.684,E2 -2058.684} C_VEL
LIN {X 0,Y 573.02,Z 345.312,A -85,B 0,C 180,E1 -2059.756,E2 -2059.756} C_VEL
LIN {X 0,Y 572.971,Z 349.676,A -85,B 0,C 180,E1 -2060.824,E2 -2060.824} C_VEL
LIN {X 0,Y 572.984,Z 351.979,A -85,B 0,C 180,E1 -2061.536,E2 -2061.536} C_VEL
LIN {X 0,Y 572.988,Z 353.839,A -85,B 0,C 180,E1 -2062.245,E2 -2062.245} C_VEL
LIN {X 0,Y 573.032,Z 355.95,A -85,B 0,C 180,E1 -2063.432,E2 -2063.432} C_VEL
LIN {X 0,Y 572.992,Z 356.803,A -85,B 0,C 180,E1 -2064.368,E2 -2064.368} C_VEL
LIN {X 0,Y 572.937,Z 356.998,A -85,B 0,C 180,E1 -2065.074,E2 -2065.074} C_VEL
LIN {X 0,Y 573.008,Z 356.765,A -85,B 0,C 180,E1 -2065.779,E2 -2065.779} C_VEL
LIN {X 0,Y 573.006,Z 356.147,A -85,B 0,C 180,E1 -2066.483,E2 -2066.483} C_VEL
LIN {X 0,Y 572.956,Z 355.143,A -85,B 0,C 180,E1 -2067.187,E2 -2067.187} C_VEL
LIN {X 0,Y 572.941,Z 353.729,A -85,B 0,C 180,E1 -2067.89,E2 -2067.89} C_VEL
LIN {X 0,Y 572.985,Z 350.794,A -85,B 0,C 180,E1 -2068.945,E2 -2068.945} C_VEL
LIN {X 0,Y 573,Z 346.83,A -85,B 0,C 180,E1 -2069.999,E2 -2069.999} C_VEL
LIN {X 0,Y 573.07,Z 341.734,A -85,B 0,C 180,E1 -2071.053,E2 -2071.053} C_VEL
LIN {X 0,Y 573.058,Z 335.34,A -85,B 0,C 180,E1 -2072.108,E2 -2072.108} C_VEL
LIN {X 0,Y 573.22,Z 327.381,A -85,B 0,C 180,E1 -2073.162,E2 -2073.162} C_VEL
LIN {X 0,Y 573.247,Z 317.519,A -85,B 0,C 180,E1 -2074.218,E2 -2074.218} C_VEL
LIN {X 0,Y 573.367,Z 307.183,A -85,B 0,C 180,E1 -2075.098,E2 -2075.098} C_VEL
LIN {X 0,Y 573.534,Z 295.562,A -85,B 0,C 180,E1 -2075.89,E2 -2075.89} C_VEL
LIN {X 0,Y 573.69,Z 283.981,A -85,B 0,C 180,E1 -2076.505,E2 -2076.505} C_VEL
LIN {X 0,Y 573.721,Z 272.31,A -85,B 0,C 180,E1 -2076.981,E2 -2076.981} C_VEL
LIN {X 0,Y 573.813,Z 259.502,A -85,B 0,C 180,E1 -2077.353,E2 -2077.353} C_VEL
LIN {X 0,Y 573.87,Z 247.545,A -85,B 0,C 180,E1 -2077.571,E2 -2077.571} C_VEL
LIN {X 0,Y 574.033,Z 151.255,A -85,B 0,C 180,E1 -2078.78,E2 -2078.78} C_VEL
LIN {X 0,Y 573.225,Z 146.654,A -85,B 0,C 180,E1 -2078.859,E2 -2078.859} C_VEL
LIN {X 0,Y 573.38,Z 131.547,A -85,B 0,C 180,E1 -2081.667,E2 -2081.667} C_VEL
LIN {X 0,Y 573.268,Z 122.076,A -85,B 0,C 180,E1 -2083.469,E2 -2083.469} C_VEL
LIN {X 0,Y 573.246,Z 122.084,A -85,B 0,C 180,E1 -2086.378,E2 -2086.378} C_VEL
LIN {X 0,Y 573.267,Z 122.071,A -85,B 0,C 180,E1 -2089.329,E2 -2089.329} C_VEL
LIN {X 0,Y 573.235,Z 122.083,A -85,B 0,C 180,E1 -2092.337,E2 -2092.337} C_VEL
LIN {X 0,Y 573.254,Z 122.074,A -85,B 0,C 180,E1 -2095.409,E2 -2095.409} C_VEL
LIN {X 0,Y 573.23,Z 122.078,A -85,B 0,C 180,E1 -2098.564,E2 -2098.564} C_VEL
LIN {X 0,Y 573.224,Z 122.077,A -85,B 0,C 180,E1 -2100.992,E2 -2100.992} C_VEL
LIN {X 0,Y 573.26,Z 122.077,A -85,B 0,C 180,E1 -2103.523,E2 -2103.523} C_VEL
LIN {X 0,Y 573.21,Z 122.083,A -85,B 0,C 180,E1 -2106.05,E2 -2106.05} C_VEL
LIN {X 0,Y 573.24,Z 122.075,A -85,B 0,C 180,E1 -2108.7,E2 -2108.7} C_VEL
LIN {X 0,Y 573.223,Z 122.086,A -85,B 0,C 180,E1 -2111.592,E2 -2111.592} C_VEL
LIN {X 0,Y 573.218,Z 122.078,A -85,B 0,C 180,E1 -2114.333,E2 -2114.333} C_VEL
LIN {X 0,Y 573.23,Z 122.085,A -85,B 0,C 180,E1 -2117.358,E2 -2117.358} C_VEL
LIN {X 0,Y 573.229,Z 122.076,A -85,B 0,C 180,E1 -2120.391,E2 -2120.391} C_VEL
LIN {X 0,Y 573.243,Z 122.082,A -85,B 0,C 180,E1 -2123.077,E2 -2123.077} C_VEL
LIN {X 0,Y 573.246,Z 122.076,A -85,B 0,C 180,E1 -2125.67,E2 -2125.67} C_VEL
LIN {X 0,Y 573.227,Z 122.077,A -85,B 0,C 180,E1 -2128.183,E2 -2128.183} C_VEL
LIN {X 0,Y 573.245,Z 122.079,A -85,B 0,C 180,E1 -2130.633,E2 -2130.633} C_VEL
LIN {X 0,Y 573.203,Z 122.087,A -85,B 0,C 180,E1 -2133.021,E2 -2133.021} C_VEL
LIN {X 0,Y 573.205,Z 122.081,A -85,B 0,C 180,E1 -2135.363,E2 -2135.363} C_VEL
LIN {X 0,Y 573.209,Z 122.079,A -85,B 0,C 180,E1 -2137.661,E2 -2137.661} C_VEL
LIN {X 0,Y 573.253,Z 122.082,A -85,B 0,C 180,E1 -2140.669,E2 -2140.669} C_VEL
LIN {X 0,Y 573.202,Z 122.08,A -85,B 0,C 180,E1 -2143.62,E2 -2143.62} C_VEL
LIN {X 0,Y 573.227,Z 122.078,A -85,B 0,C 180,E1 -2145.806,E2 -2145.806} C_VEL
LIN {X 0,Y 573.25,Z 122.078,A -85,B 0,C 180,E1 -2148.745,E2 -2148.745} C_VEL
LIN {X 0,Y 573.231,Z 122.077,A -85,B 0,C 180,E1 -2151.54,E2 -2151.54} C_VEL
LIN {X 0,Y 573.266,Z 122.078,A -85,B 0,C 180,E1 -2154.371,E2 -2154.371} C_VEL
LIN {X 0,Y 573.3,Z 122.075,A -85,B 0,C 180,E1 -2157.892,E2 -2157.892} C_VEL
LIN {X 0,Y 573.305,Z 122.075,A -85,B 0,C 180,E1 -2160,E2 -2160} C_VEL
LIN {X 0,Y 573.26,Z 122.073,A -85,B 0,C 180,E1 -2162.811,E2 -2162.811} C_VEL
LIN {X 0,Y 573.268,Z 122.079,A -85,B 0,C 180,E1 -2165.628,E2 -2165.628} C_VEL
LIN {X 0,Y 573.232,Z 122.077,A -85,B 0,C 180,E1 -2168.46,E2 -2168.46} C_VEL
LIN {X 0,Y 573.259,Z 122.078,A -85,B 0,C 180,E1 -2171.312,E2 -2171.312} C_VEL
LIN {X 0,Y 573.241,Z 122.075,A -85,B 0,C 180,E1 -2174.414,E2 -2174.414} C_VEL
LIN {X 0,Y 573.233,Z 122.081,A -85,B 0,C 180,E1 -2177.112,E2 -2177.112} C_VEL
LIN {X 0,Y 573.221,Z 122.078,A -85,B 0,C 180,E1 -2180.078,E2 -2180.078} C_VEL
LIN {X 0,Y 573.209,Z 122.079,A -85,B 0,C 180,E1 -2182.339,E2 -2182.339} C_VEL
LIN {X 0,Y 573.224,Z 122.083,A -85,B 0,C 180,E1 -2185.412,E2 -2185.412} C_VEL
LIN {X 0,Y 573.236,Z 122.076,A -85,B 0,C 180,E1 -2188.029,E2 -2188.029} C_VEL
LIN {X 0,Y 573.217,Z 122.086,A -85,B 0,C 180,E1 -2190.883,E2 -2190.883} C_VEL
LIN {X 0,Y 573.231,Z 122.077,A -85,B 0,C 180,E1 -2193.521,E2 -2193.521} C_VEL
LIN {X 0,Y 573.205,Z 122.08,A -85,B 0,C 180,E1 -2196.052,E2 -2196.052} C_VEL
LIN {X 0,Y 573.232,Z 122.085,A -85,B 0,C 180,E1 -2198.702,E2 -2198.702} C_VEL
LIN {X 0,Y 573.219,Z 122.077,A -85,B 0,C 180,E1 -2201.594,E2 -2201.594} C_VEL
LIN {X 0,Y 573.225,Z 122.083,A -85,B 0,C 180,E1 -2204.335,E2 -2204.335} C_VEL
LIN {X 0,Y 573.233,Z 122.076,A -85,B 0,C 180,E1 -2207.36,E2 -2207.36} C_VEL
LIN {X 0,Y 573.245,Z 122.08,A -85,B 0,C 180,E1 -2210.568,E2 -2210.568} C_VEL
LIN {X 0,Y 573.247,Z 122.074,A -85,B 0,C 180,E1 -2213.079,E2 -2213.079} C_VEL
LIN {X 0,Y 573.261,Z 122.075,A -85,B 0,C 180,E1 -2215.672,E2 -2215.672} C_VEL
LIN {X 0,Y 573.243,Z 122.083,A -85,B 0,C 180,E1 -2218.186,E2 -2218.186} C_VEL
LIN {X 0,Y 573.259,Z 122.074,A -85,B 0,C 180,E1 -2220.635,E2 -2220.635} C_VEL
LIN {X 0,Y 573.248,Z 122.074,A -85,B 0,C 180,E1 -2223.025,E2 -2223.025} C_VEL
LIN {X 0,Y 573.274,Z 122.073,A -85,B 0,C 180,E1 -2225.367,E2 -2225.367} C_VEL
LIN {X 0,Y 573.271,Z 122.238,A -85,B 0,C 180,E1 -2226.181,E2 -2226.181} C_VEL
LIN {X 0,Y 573.999,Z 127.389,A -85,B 0,C 180,E1 -2226.934,E2 -2226.934} C_VEL
LIN {X 0,Y 573.845,Z 146.398,A -85,B 0,C 180,E1 -2229.572,E2 -2229.572} C_VEL
LIN {X 0,Y 573.656,Z 166.823,A -85,B 0,C 180,E1 -2232.368,E2 -2232.368} C_VEL
LIN {X 0,Y 573.449,Z 186.634,A -85,B 0,C 180,E1 -2235.087,E2 -2235.087} C_VEL
LIN {X 0,Y 573.411,Z 194.528,A -85,B 0,C 180,E1 -2236.162,E2 -2236.162} C_VEL
LIN {X 0,Y 574.058,Z 200.576,A -85,B 0,C 180,E1 -2236.257,E2 -2236.257} C_VEL
LIN {X 0,Y 573.849,Z 302.989,A -85,B 0,C 180,E1 -2237.558,E2 -2237.558} C_VEL
LIN {X 0,Y 573.777,Z 316.246,A -85,B 0,C 180,E1 -2237.87,E2 -2237.87} C_VEL
LIN {X 0,Y 573.691,Z 328.397,A -85,B 0,C 180,E1 -2238.295,E2 -2238.295} C_VEL
LIN {X 0,Y 573.608,Z 340.64,A -85,B 0,C 180,E1 -2238.874,E2 -2238.874} C_VEL
LIN {X 0,Y 573.427,Z 352.21,A -85,B 0,C 180,E1 -2239.586,E2 -2239.586} C_VEL
LIN {X 0,Y 573.332,Z 362.612,A -85,B 0,C 180,E1 -2240.386,E2 -2240.386} C_VEL
LIN {X 0,Y 573.24,Z 371.121,A -85,B 0,C 180,E1 -2241.185,E2 -2241.185} C_VEL
LIN {X 0,Y 573.16,Z 378.967,A -85,B 0,C 180,E1 -2242.072,E2 -2242.072} C_VEL
LIN {X 0,Y 573.073,Z 386.585,A -85,B 0,C 180,E1 -2243.127,E2 -2243.127} C_VEL
LIN {X 0,Y 573.07,Z 393.684,A -85,B 0,C 180,E1 -2244.37,E2 -2244.37} C_VEL
LIN {X 0,Y 573.028,Z 398.375,A -85,B 0,C 180,E1 -2245.428,E2 -2245.428} C_VEL
LIN {X 0,Y 573.022,Z 401.96,A -85,B 0,C 180,E1 -2246.485,E2 -2246.485} C_VEL
LIN {X 0,Y 572.959,Z 403.809,A -85,B 0,C 180,E1 -2247.188,E2 -2247.188} C_VEL
LIN {X 0,Y 572.946,Z 406.186,A -85,B 0,C 180,E1 -2248.595,E2 -2248.595} C_VEL
LIN {X 0,Y 572.938,Z 407,A -85,B 0,C 180,E1 -2250.001,E2 -2250.001} C_VEL
LIN {X 0,Y 572.946,Z 406.185,A -85,B 0,C 180,E1 -2251.406,E2 -2251.406} C_VEL
LIN {X 0,Y 572.94,Z 405.198,A -85,B 0,C 180,E1 -2252.11,E2 -2252.11} C_VEL
LIN {X 0,Y 572.959,Z 403.809,A -85,B 0,C 180,E1 -2252.813,E2 -2252.813} C_VEL
LIN {X 0,Y 573.015,Z 400.894,A -85,B 0,C 180,E1 -2253.869,E2 -2253.869} C_VEL
LIN {X 0,Y 572.963,Z 396.946,A -85,B 0,C 180,E1 -2254.926,E2 -2254.926} C_VEL
LIN {X 0,Y 573.065,Z 390.873,A -85,B 0,C 180,E1 -2256.161,E2 -2256.161} C_VEL
LIN {X 0,Y 573.12,Z 384.233,A -85,B 0,C 180,E1 -2257.221,E2 -2257.221} C_VEL
LIN {X 0,Y 573.201,Z 375.987,A -85,B 0,C 180,E1 -2258.284,E2 -2258.284} C_VEL
LIN {X 0,Y 573.287,Z 367.533,A -85,B 0,C 180,E1 -2259.171,E2 -2259.171} C_VEL
LIN {X 0,Y 573.427,Z 357.089,A -85,B 0,C 180,E1 -2260.059,E2 -2260.059} C_VEL
LIN {X 0,Y 573.544,Z 345.424,A -85,B 0,C 180,E1 -2260.853,E2 -2260.853} C_VEL
LIN {X 0,Y 573.652,Z 334.298,A -85,B 0,C 180,E1 -2261.447,E2 -2261.447} C_VEL
LIN {X 0,Y 573.759,Z 321.155,A -85,B 0,C 180,E1 -2261.974,E2 -2261.974} C_VEL
LIN {X 0,Y 573.843,Z 308.497,A -85,B 0,C 180,E1 -2262.332,E2 -2262.332} C_VEL
